DATA_BLOCK "DB_EmXcut_M203_SnapM201_HMI"
{ DB_Accessible_From_OPC_UA := 'FALSE' ;
 DB_Accessible_From_Webserver := 'FALSE' ;
 S7_Optimized_Access := 'FALSE' }
VERSION : 0.1
NON_RETAIN
   STRUCT
      tALM { ExternalWritable := 'False'} : Struct   // HMI Alarms
         tE { ExternalWritable := 'False'} : Struct   // Stopping faults
            xSpare_0 { ExternalWritable := 'False'} : Bool;
            xSpare_1 { ExternalWritable := 'False'} : Bool;
            xSpare_2 { ExternalWritable := 'False'} : Bool;
            xSpare_3 { ExternalWritable := 'False'} : Bool;
            xSpare_4 { ExternalWritable := 'False'} : Bool;
            xSpare_5 { ExternalWritable := 'False'} : Bool;
            xSpare_6 { ExternalWritable := 'False'} : Bool;
            xSpare_7 { ExternalWritable := 'False'} : Bool;
            xSpare_8 { ExternalWritable := 'False'} : Bool;
            xSpare_9 { ExternalWritable := 'False'} : Bool;
            xSpare_10 { ExternalWritable := 'False'} : Bool;
            xSpare_11 { ExternalWritable := 'False'} : Bool;
            xSpare_12 { ExternalWritable := 'False'} : Bool;
            xSpare_13 { ExternalWritable := 'False'} : Bool;
            xSpare_14 { ExternalWritable := 'False'} : Bool;
            xSpare_15 { ExternalWritable := 'False'} : Bool;
            xSpare_16 { ExternalWritable := 'False'} : Bool;
            xSpare_17 { ExternalWritable := 'False'} : Bool;
            xSpare_18 { ExternalWritable := 'False'} : Bool;
            xSpare_19 { ExternalWritable := 'False'} : Bool;
            xSpare_20 { ExternalWritable := 'False'} : Bool;
            xSpare_21 { ExternalWritable := 'False'} : Bool;
            xSpare_22 { ExternalWritable := 'False'} : Bool;
            xSpare_23 { ExternalWritable := 'False'} : Bool;
            xSpare_24 { ExternalWritable := 'False'} : Bool;
            xSpare_25 { ExternalWritable := 'False'} : Bool;
            xSpare_26 { ExternalWritable := 'False'} : Bool;
            xSpare_27 { ExternalWritable := 'False'} : Bool;
            xSpare_28 { ExternalWritable := 'False'} : Bool;
            xSpare_29 { ExternalWritable := 'False'} : Bool;
            xSpare_30 { ExternalWritable := 'False'} : Bool;
            xSpare_31 { ExternalWritable := 'False'} : Bool;
         END_STRUCT;
         tS { ExternalWritable := 'False'} : Struct   // Stopping faults
            xMachineNotReady { ExternalWritable := 'False'} : Bool;   // Machine not ready
            xQMProtection { ExternalWritable := 'False'} : Bool;   // A172QM1.Protection
            xSpare_2 { ExternalAccessible := 'False'; ExternalVisible := 'False'; ExternalWritable := 'False'} : Bool;
            xSpare_3 { ExternalAccessible := 'False'; ExternalVisible := 'False'; ExternalWritable := 'False'} : Bool;
            xSpare_4 { ExternalAccessible := 'False'; ExternalVisible := 'False'; ExternalWritable := 'False'} : Bool;
            xSpare_5 { ExternalAccessible := 'False'; ExternalVisible := 'False'; ExternalWritable := 'False'} : Bool;
            xSpare_6 { ExternalAccessible := 'False'; ExternalVisible := 'False'; ExternalWritable := 'False'} : Bool;
            xSpare_7 { ExternalAccessible := 'False'; ExternalVisible := 'False'; ExternalWritable := 'False'} : Bool;
            xSpare_8 { ExternalAccessible := 'False'; ExternalVisible := 'False'; ExternalWritable := 'False'} : Bool;
            xSpare_9 { ExternalAccessible := 'False'; ExternalVisible := 'False'; ExternalWritable := 'False'} : Bool;
            xSpare_10 { ExternalAccessible := 'False'; ExternalVisible := 'False'; ExternalWritable := 'False'} : Bool;
            xSpare_11 { ExternalAccessible := 'False'; ExternalVisible := 'False'; ExternalWritable := 'False'} : Bool;
            xSpare_12 { ExternalAccessible := 'False'; ExternalVisible := 'False'; ExternalWritable := 'False'} : Bool;
            xSpare_13 { ExternalAccessible := 'False'; ExternalVisible := 'False'; ExternalWritable := 'False'} : Bool;
            xSpare_14 { ExternalAccessible := 'False'; ExternalVisible := 'False'; ExternalWritable := 'False'} : Bool;
            xSpare_15 { ExternalAccessible := 'False'; ExternalVisible := 'False'; ExternalWritable := 'False'} : Bool;
            xSpare_16 { ExternalAccessible := 'False'; ExternalVisible := 'False'; ExternalWritable := 'False'} : Bool;
            xSpare_17 { ExternalAccessible := 'False'; ExternalVisible := 'False'; ExternalWritable := 'False'} : Bool;
            xSpare_18 { ExternalAccessible := 'False'; ExternalVisible := 'False'; ExternalWritable := 'False'} : Bool;
            xSpare_19 { ExternalAccessible := 'False'; ExternalVisible := 'False'; ExternalWritable := 'False'} : Bool;
            xSpare_20 { ExternalAccessible := 'False'; ExternalVisible := 'False'; ExternalWritable := 'False'} : Bool;
            xSpare_21 { ExternalAccessible := 'False'; ExternalVisible := 'False'; ExternalWritable := 'False'} : Bool;
            xSpare_22 { ExternalAccessible := 'False'; ExternalVisible := 'False'; ExternalWritable := 'False'} : Bool;
            xSpare_23 { ExternalAccessible := 'False'; ExternalVisible := 'False'; ExternalWritable := 'False'} : Bool;
            xSpare_24 { ExternalAccessible := 'False'; ExternalVisible := 'False'; ExternalWritable := 'False'} : Bool;
            xSpare_25 { ExternalAccessible := 'False'; ExternalVisible := 'False'; ExternalWritable := 'False'} : Bool;
            xSpare_26 { ExternalAccessible := 'False'; ExternalVisible := 'False'; ExternalWritable := 'False'} : Bool;
            xSpare_27 { ExternalAccessible := 'False'; ExternalVisible := 'False'; ExternalWritable := 'False'} : Bool;
            xSpare_28 { ExternalAccessible := 'False'; ExternalVisible := 'False'; ExternalWritable := 'False'} : Bool;
            xSpare_29 { ExternalAccessible := 'False'; ExternalVisible := 'False'; ExternalWritable := 'False'} : Bool;
            xSpare_30 { ExternalAccessible := 'False'; ExternalVisible := 'False'; ExternalWritable := 'False'} : Bool;
            xSpare_31 { ExternalAccessible := 'False'; ExternalVisible := 'False'; ExternalWritable := 'False'} : Bool;
         END_STRUCT;
         tF { ExternalAccessible := 'False'; ExternalVisible := 'False'; ExternalWritable := 'False'} : Struct   // Faults
            xSpare_0 { ExternalAccessible := 'False'; ExternalVisible := 'False'; ExternalWritable := 'False'} : Bool;
            xSpare_1 { ExternalAccessible := 'False'; ExternalVisible := 'False'; ExternalWritable := 'False'} : Bool;
            xSpare_2 { ExternalAccessible := 'False'; ExternalVisible := 'False'; ExternalWritable := 'False'} : Bool;
            xSpare_3 { ExternalAccessible := 'False'; ExternalVisible := 'False'; ExternalWritable := 'False'} : Bool;
            xSpare_4 { ExternalAccessible := 'False'; ExternalVisible := 'False'; ExternalWritable := 'False'} : Bool;
            xSpare_5 { ExternalAccessible := 'False'; ExternalVisible := 'False'; ExternalWritable := 'False'} : Bool;
            xSpare_6 { ExternalAccessible := 'False'; ExternalVisible := 'False'; ExternalWritable := 'False'} : Bool;
            xSpare_7 { ExternalAccessible := 'False'; ExternalVisible := 'False'; ExternalWritable := 'False'} : Bool;
            xSpare_8 { ExternalAccessible := 'False'; ExternalVisible := 'False'; ExternalWritable := 'False'} : Bool;
            xSpare_9 { ExternalAccessible := 'False'; ExternalVisible := 'False'; ExternalWritable := 'False'} : Bool;
            xSpare_10 { ExternalAccessible := 'False'; ExternalVisible := 'False'; ExternalWritable := 'False'} : Bool;
            xSpare_11 { ExternalAccessible := 'False'; ExternalVisible := 'False'; ExternalWritable := 'False'} : Bool;
            xSpare_12 { ExternalAccessible := 'False'; ExternalVisible := 'False'; ExternalWritable := 'False'} : Bool;
            xSpare_13 { ExternalAccessible := 'False'; ExternalVisible := 'False'; ExternalWritable := 'False'} : Bool;
            xSpare_14 { ExternalAccessible := 'False'; ExternalVisible := 'False'; ExternalWritable := 'False'} : Bool;
            xSpare_15 { ExternalAccessible := 'False'; ExternalVisible := 'False'; ExternalWritable := 'False'} : Bool;
            xSpare_16 { ExternalAccessible := 'False'; ExternalVisible := 'False'; ExternalWritable := 'False'} : Bool;
            xSpare_17 { ExternalAccessible := 'False'; ExternalVisible := 'False'; ExternalWritable := 'False'} : Bool;
            xSpare_18 { ExternalAccessible := 'False'; ExternalVisible := 'False'; ExternalWritable := 'False'} : Bool;
            xSpare_19 { ExternalAccessible := 'False'; ExternalVisible := 'False'; ExternalWritable := 'False'} : Bool;
            xSpare_20 { ExternalAccessible := 'False'; ExternalVisible := 'False'; ExternalWritable := 'False'} : Bool;
            xSpare_21 { ExternalAccessible := 'False'; ExternalVisible := 'False'; ExternalWritable := 'False'} : Bool;
            xSpare_22 { ExternalAccessible := 'False'; ExternalVisible := 'False'; ExternalWritable := 'False'} : Bool;
            xSpare_23 { ExternalAccessible := 'False'; ExternalVisible := 'False'; ExternalWritable := 'False'} : Bool;
            xSpare_24 { ExternalAccessible := 'False'; ExternalVisible := 'False'; ExternalWritable := 'False'} : Bool;
            xSpare_25 { ExternalAccessible := 'False'; ExternalVisible := 'False'; ExternalWritable := 'False'} : Bool;
            xSpare_26 { ExternalAccessible := 'False'; ExternalVisible := 'False'; ExternalWritable := 'False'} : Bool;
            xSpare_27 { ExternalAccessible := 'False'; ExternalVisible := 'False'; ExternalWritable := 'False'} : Bool;
            xSpare_28 { ExternalAccessible := 'False'; ExternalVisible := 'False'; ExternalWritable := 'False'} : Bool;
            xSpare_29 { ExternalAccessible := 'False'; ExternalVisible := 'False'; ExternalWritable := 'False'} : Bool;
            xSpare_30 { ExternalAccessible := 'False'; ExternalVisible := 'False'; ExternalWritable := 'False'} : Bool;
            xSpare_31 { ExternalAccessible := 'False'; ExternalVisible := 'False'; ExternalWritable := 'False'} : Bool;
         END_STRUCT;
         tW { ExternalAccessible := 'False'; ExternalVisible := 'False'; ExternalWritable := 'False'} : Struct   // Warnings
            xSpare_0 { ExternalAccessible := 'False'; ExternalVisible := 'False'; ExternalWritable := 'False'} : Bool;
            xSpare_1 { ExternalAccessible := 'False'; ExternalVisible := 'False'; ExternalWritable := 'False'} : Bool;
            xSpare_2 { ExternalAccessible := 'False'; ExternalVisible := 'False'; ExternalWritable := 'False'} : Bool;
            xSpare_3 { ExternalAccessible := 'False'; ExternalVisible := 'False'; ExternalWritable := 'False'} : Bool;
            xSpare_4 { ExternalAccessible := 'False'; ExternalVisible := 'False'; ExternalWritable := 'False'} : Bool;
            xSpare_5 { ExternalAccessible := 'False'; ExternalVisible := 'False'; ExternalWritable := 'False'} : Bool;
            xSpare_6 { ExternalAccessible := 'False'; ExternalVisible := 'False'; ExternalWritable := 'False'} : Bool;
            xSpare_7 { ExternalAccessible := 'False'; ExternalVisible := 'False'; ExternalWritable := 'False'} : Bool;
            xSpare_8 { ExternalAccessible := 'False'; ExternalVisible := 'False'; ExternalWritable := 'False'} : Bool;
            xSpare_9 { ExternalAccessible := 'False'; ExternalVisible := 'False'; ExternalWritable := 'False'} : Bool;
            xSpare_10 { ExternalAccessible := 'False'; ExternalVisible := 'False'; ExternalWritable := 'False'} : Bool;
            xSpare_11 { ExternalAccessible := 'False'; ExternalVisible := 'False'; ExternalWritable := 'False'} : Bool;
            xSpare_12 { ExternalAccessible := 'False'; ExternalVisible := 'False'; ExternalWritable := 'False'} : Bool;
            xSpare_13 { ExternalAccessible := 'False'; ExternalVisible := 'False'; ExternalWritable := 'False'} : Bool;
            xSpare_14 { ExternalAccessible := 'False'; ExternalVisible := 'False'; ExternalWritable := 'False'} : Bool;
            xSpare_15 { ExternalAccessible := 'False'; ExternalVisible := 'False'; ExternalWritable := 'False'} : Bool;
            xSpare_16 { ExternalAccessible := 'False'; ExternalVisible := 'False'; ExternalWritable := 'False'} : Bool;
            xSpare_17 { ExternalAccessible := 'False'; ExternalVisible := 'False'; ExternalWritable := 'False'} : Bool;
            xSpare_18 { ExternalAccessible := 'False'; ExternalVisible := 'False'; ExternalWritable := 'False'} : Bool;
            xSpare_19 { ExternalAccessible := 'False'; ExternalVisible := 'False'; ExternalWritable := 'False'} : Bool;
            xSpare_20 { ExternalAccessible := 'False'; ExternalVisible := 'False'; ExternalWritable := 'False'} : Bool;
            xSpare_21 { ExternalAccessible := 'False'; ExternalVisible := 'False'; ExternalWritable := 'False'} : Bool;
            xSpare_22 { ExternalAccessible := 'False'; ExternalVisible := 'False'; ExternalWritable := 'False'} : Bool;
            xSpare_23 { ExternalAccessible := 'False'; ExternalVisible := 'False'; ExternalWritable := 'False'} : Bool;
            xSpare_24 { ExternalAccessible := 'False'; ExternalVisible := 'False'; ExternalWritable := 'False'} : Bool;
            xSpare_25 { ExternalAccessible := 'False'; ExternalVisible := 'False'; ExternalWritable := 'False'} : Bool;
            xSpare_26 { ExternalAccessible := 'False'; ExternalVisible := 'False'; ExternalWritable := 'False'} : Bool;
            xSpare_27 { ExternalAccessible := 'False'; ExternalVisible := 'False'; ExternalWritable := 'False'} : Bool;
            xSpare_28 { ExternalAccessible := 'False'; ExternalVisible := 'False'; ExternalWritable := 'False'} : Bool;
            xSpare_29 { ExternalAccessible := 'False'; ExternalVisible := 'False'; ExternalWritable := 'False'} : Bool;
            xSpare_30 { ExternalAccessible := 'False'; ExternalVisible := 'False'; ExternalWritable := 'False'} : Bool;
            xSpare_31 { ExternalAccessible := 'False'; ExternalVisible := 'False'; ExternalWritable := 'False'} : Bool;
         END_STRUCT;
      END_STRUCT;
      tHMR { ExternalWritable := 'False'} : Struct   // HMI Read
         xSpare0 { ExternalWritable := 'False'} : Bool;   //
         xSpare1 { ExternalWritable := 'False'} : Bool;   //
         xSpare2 { ExternalWritable := 'False'} : Bool;
         xSpare3 { ExternalWritable := 'False'} : Bool;
         xSpare4 { ExternalWritable := 'False'} : Bool;
         xSpare5 { ExternalWritable := 'False'} : Bool;
         xSpare6 { ExternalWritable := 'False'} : Bool;
         xSpare7 { ExternalWritable := 'False'} : Bool;
         xSpare8 { ExternalWritable := 'False'} : Bool;
         xSpare9 { ExternalWritable := 'False'} : Bool;
         xSpare10 { ExternalWritable := 'False'} : Bool;
         xSpare11 { ExternalWritable := 'False'} : Bool;
         xSpare12 { ExternalWritable := 'False'} : Bool;
         xSpare13 { ExternalWritable := 'False'} : Bool;
         xSpare14 { ExternalWritable := 'False'} : Bool;
         xSpare15 { ExternalWritable := 'False'} : Bool;
         xSpare16 { ExternalWritable := 'False'} : Bool;
         xSpare17 { ExternalWritable := 'False'} : Bool;
         xSpare18 { ExternalWritable := 'False'} : Bool;
         xSpare19 { ExternalWritable := 'False'} : Bool;
         xSpare20 { ExternalWritable := 'False'} : Bool;
         xSpare21 { ExternalWritable := 'False'} : Bool;
         xSpare22 { ExternalWritable := 'False'} : Bool;
         xSpare23 { ExternalWritable := 'False'} : Bool;
         xSpare24 { ExternalWritable := 'False'} : Bool;
         xSpare25 { ExternalWritable := 'False'} : Bool;
         xSpare26 { ExternalWritable := 'False'} : Bool;
         xSpare27 { ExternalWritable := 'False'} : Bool;
         xSpare28 { ExternalWritable := 'False'} : Bool;
         xSpare29 { ExternalWritable := 'False'} : Bool;
         xSpare30 { ExternalWritable := 'False'} : Bool;
         xSpare31 { ExternalWritable := 'False'} : Bool;
         xSpare { ExternalWritable := 'False'} : Array[0..15] of Bool;
         iSpare0 { ExternalWritable := 'False'} : Int;
         iSpare1 { ExternalWritable := 'False'} : Int;
         iSpare2 { ExternalWritable := 'False'} : Int;
         iSpare3 { ExternalWritable := 'False'} : Int;
         iSpare4 { ExternalWritable := 'False'} : Int;
         iSpare5 { ExternalWritable := 'False'} : Int;
         iSpare6 { ExternalWritable := 'False'} : Int;
         iSpare7 { ExternalWritable := 'False'} : Int;
         iSpare8 { ExternalWritable := 'False'} : Int;
         iSpare9 { ExternalWritable := 'False'} : Int;
         iSpare10 { ExternalWritable := 'False'} : Int;
         iSpare11 { ExternalWritable := 'False'} : Int;
         iSpare12 { ExternalWritable := 'False'} : Int;
         iSpare13 { ExternalWritable := 'False'} : Int;
         iSpare14 { ExternalWritable := 'False'} : Int;
         iSpare15 { ExternalWritable := 'False'} : Int;
         iSpare16 { ExternalWritable := 'False'} : Int;
         dDistanceSnaproll_cmm { ExternalWritable := 'False'} : DInt;   // Distance from snaproll [mm/100] {mm/100|mm|x|x|M}
         dState { ExternalWritable := 'False'} : DInt;   // State  (1=No anomaly, 3=Run, 7=Anomaly) {x|x|x|x|O}
         dSpare2 { ExternalWritable := 'False'} : DInt;   //
         dSpare3 { ExternalWritable := 'False'} : DInt;
         dSpare4 { ExternalWritable := 'False'} : DInt;
         dSpare5 { ExternalWritable := 'False'} : DInt;
         dSpare6 { ExternalWritable := 'False'} : DInt;
         dSpare7 { ExternalWritable := 'False'} : DInt;
         dSpare8 { ExternalWritable := 'False'} : DInt;
         dSpare9 { ExternalWritable := 'False'} : DInt;
         dSpare10 { ExternalWritable := 'False'} : DInt;
         dSpare11 { ExternalWritable := 'False'} : DInt;
         dSpare12 { ExternalWritable := 'False'} : DInt;
         dSpare13 { ExternalWritable := 'False'} : DInt;
         dSpare14 { ExternalWritable := 'False'} : DInt;
         dSpare15 { ExternalWritable := 'False'} : DInt;
         rSpare0 { ExternalWritable := 'False'} : Real;
         rSpare1 { ExternalWritable := 'False'} : Real;
         rSpare2 { ExternalWritable := 'False'} : Real;
         rSpare3 { ExternalWritable := 'False'} : Real;
         rSpare4 { ExternalWritable := 'False'} : Real;
         rSpare5 { ExternalWritable := 'False'} : Real;
         rSpare6 { ExternalWritable := 'False'} : Real;
         rSpare7 { ExternalWritable := 'False'} : Real;
         rSpare8 { ExternalWritable := 'False'} : Real;
         tManCmd { ExternalWritable := 'False'} : Struct
            xSpare0 { ExternalWritable := 'False'} : Bool;   //
            xSpare1 { ExternalWritable := 'False'} : Bool;   //
            xSpare2 { ExternalWritable := 'False'} : Bool;
            xSpare3 { ExternalWritable := 'False'} : Bool;
            xSpare4 { ExternalWritable := 'False'} : Bool;
            xSpare5 { ExternalWritable := 'False'} : Bool;
            xSpare6 { ExternalWritable := 'False'} : Bool;
            xSpare7 { ExternalWritable := 'False'} : Bool;
            xSpare8 { ExternalWritable := 'False'} : Bool;
            xSpare9 { ExternalWritable := 'False'} : Bool;
            xSpare10 { ExternalWritable := 'False'} : Bool;
            xSpare11 { ExternalWritable := 'False'} : Bool;
            xSpare12 { ExternalWritable := 'False'} : Bool;
            xSpare13 { ExternalWritable := 'False'} : Bool;
            xSpare14 { ExternalWritable := 'False'} : Bool;
            xSpare15 { ExternalWritable := 'False'} : Bool;
            xSpare { ExternalWritable := 'False'} : Array[0..15] of Bool;
         END_STRUCT;
      END_STRUCT;
      tHMW : Struct   // HMI Write
         xSpare0 : Bool;   //
         xSpare1 : Bool;   //
         xSpare2 : Bool;   //
         xSpare3 : Bool;   //
         xSpare4 : Bool;   //
         xSpare5 : Bool;
         xSpare6 : Bool;
         xSpare7 : Bool;
         xSpare8 : Bool;   //
         xSpare9 : Bool;
         xSpare10 : Bool;
         xSpare11 : Bool;
         xSpare12 : Bool;
         xSpare13 : Bool;
         xSpare14 : Bool;   //
         xUpdateDistanceSnaproll : Bool;   // Update distance from snaproll {x|x|x|x|M}
         xSpare16 : Bool;   //
         xSpare17 : Bool;
         xSpare18 : Bool;
         xSpare19 : Bool;
         xSpare20 : Bool;
         xSpare21 : Bool;
         xSpare22 : Bool;
         xSpare23 : Bool;
         xSpare24 : Bool;
         xSpare25 : Bool;
         xSpare26 : Bool;
         xSpare27 : Bool;
         xSpare28 : Bool;
         xSpare29 : Bool;
         xSpare30 : Bool;
         xSpare31 : Bool;
         xSpare : Array[0..15] of Bool;
         iSpare0 : Int;
         iSpare1 : Int;
         iSpare2 : Int;
         iSpare3 : Int;
         iSpare4 : Int;
         iSpare5 : Int;
         iSpare6 : Int;
         iSpare7 : Int;
         iSpare8 : Int;
         iSpare9 : Int;
         iSpare10 : Int;
         iSpare11 : Int;
         iSpare12 : Int;
         iSpare13 : Int;
         iSpare14 : Int;
         iSpare15 : Int;
         iSpare16 : Int;
         dDistanceSnaproll_cmm : DInt;   // Distance from snaproll [mm/100] {mm/100|mm|1|70000|M}
         dSnapDuration_ms : DInt;   // Time snap in up position [ms] {ms|s|0|1|O}
         AccelerationDelay_ms : DInt;   // Acceleration delay [ms] {ms|s|0|1|O}
         dSpare3 : DInt;
         dSpare4 : DInt;
         dSpare5 : DInt;
         dSpare6 : DInt;
         dSpare7 : DInt;
         dSpare8 : DInt;
         dSpare9 : DInt;
         dSpare10 : DInt;
         dSpare11 : DInt;
         dSpare12 : DInt;
         dSpare13 : DInt;
         dSpare14 : DInt;
         dSpare15 : DInt;
         dSpare16 : DInt;
         rPlateLenght_mm : Real;   // Maximum plate lenght for contrast enabling [mm] {mm|mm|1|7000|O}
         rBreakPosOffset_mm : Real;   // BreakOffset [mm] {mm|mm|1|1000|O}
         rSpare2 : Real;
         rSpare3 : Real;
         rSpare4 : Real;
         rSpare5 : Real;
         rSpare6 : Real;
         rSpare7 : Real;
         rSpare8 : Real;
         tManCmd : Struct
            xSpare0 : Bool;
            xSpare1 : Bool;   //
            xSpare2 { ExternalWritable := 'False'} : Bool;
            xSpare3 { ExternalWritable := 'False'} : Bool;
            xSpare4 { ExternalWritable := 'False'} : Bool;
            xSpare5 { ExternalWritable := 'False'} : Bool;
            xSpare6 { ExternalWritable := 'False'} : Bool;
            xSpare7 { ExternalWritable := 'False'} : Bool;
            xSpare8 { ExternalWritable := 'False'} : Bool;
            xSpare9 { ExternalWritable := 'False'} : Bool;
            xSpare10 { ExternalWritable := 'False'} : Bool;
            xSpare11 { ExternalWritable := 'False'} : Bool;
            xSpare12 { ExternalWritable := 'False'} : Bool;
            xSpare13 { ExternalWritable := 'False'} : Bool;
            xSpare14 { ExternalWritable := 'False'} : Bool;
            xSpare15 { ExternalWritable := 'False'} : Bool;
            xSpare16 : Bool;
            xSpare17 : Bool;
            xSpare18 : Bool;
            xSpare19 : Bool;
            xSpare20 : Bool;
            xSpare21 : Bool;
            xSpare22 : Bool;
            xSpare23 : Bool;
            xSpare24 : Bool;
            xSpare25 : Bool;
            xSpare26 : Bool;
            xSpare27 : Bool;
            xSpare28 : Bool;
            xSpare29 : Bool;
            xSpare30 : Bool;
            xSpare31 : Bool;
         END_STRUCT;
      END_STRUCT;
   END_STRUCT;


BEGIN
   tHMW.tManCmd.xSpare0 := false;
   tHMW.tManCmd.xSpare1 := false;

END_DATA_BLOCK

DATA_BLOCK "DB_Oil_Manager_HMI"
{ DB_Accessible_From_OPC_UA := 'FALSE' ;
 DB_Accessible_From_Webserver := 'FALSE' ;
 S7_Optimized_Access := 'FALSE' }
VERSION : 0.1
   STRUCT
      tALM { ExternalWritable := 'False'} : Struct   // HMI Alarms
         tE { ExternalWritable := 'False'} : Struct   // Stopping faults
            xSpare_0 { ExternalWritable := 'False'} : Bool;
            xSpare_1 { ExternalWritable := 'False'} : Bool;
            xSpare_2 { ExternalWritable := 'False'} : Bool;
            xSpare_3 { ExternalWritable := 'False'} : Bool;
            xSpare_4 { ExternalWritable := 'False'} : Bool;
            xSpare_5 { ExternalWritable := 'False'} : Bool;
            xSpare_6 { ExternalWritable := 'False'} : Bool;
            xSpare_7 { ExternalWritable := 'False'} : Bool;
            xSpare_8 { ExternalWritable := 'False'} : Bool;
            xSpare_9 { ExternalWritable := 'False'} : Bool;
            xSpare_10 { ExternalWritable := 'False'} : Bool;
            xSpare_11 { ExternalWritable := 'False'} : Bool;
            xSpare_12 { ExternalWritable := 'False'} : Bool;
            xSpare_13 { ExternalWritable := 'False'} : Bool;
            xSpare_14 { ExternalWritable := 'False'} : Bool;
            xSpare_15 { ExternalWritable := 'False'} : Bool;
            xSpare_16 { ExternalWritable := 'False'} : Bool;
            xSpare_17 { ExternalWritable := 'False'} : Bool;
            xSpare_18 { ExternalWritable := 'False'} : Bool;
            xSpare_19 { ExternalWritable := 'False'} : Bool;
            xSpare_20 { ExternalWritable := 'False'} : Bool;
            xSpare_21 { ExternalWritable := 'False'} : Bool;
            xSpare_22 { ExternalWritable := 'False'} : Bool;
            xSpare_23 { ExternalWritable := 'False'} : Bool;
            xSpare_24 { ExternalWritable := 'False'} : Bool;
            xSpare_25 { ExternalWritable := 'False'} : Bool;
            xSpare_26 { ExternalWritable := 'False'} : Bool;
            xSpare_27 { ExternalWritable := 'False'} : Bool;
            xSpare_28 { ExternalWritable := 'False'} : Bool;
            xSpare_29 { ExternalWritable := 'False'} : Bool;
            xSpare_30 { ExternalWritable := 'False'} : Bool;
            xSpare_31 { ExternalWritable := 'False'} : Bool;
         END_STRUCT;
         tS { ExternalWritable := 'False'} : Struct   // Stopping faults machine
            xPowerSupplyControl { ExternalWritable := 'False'} : Bool;   // L+.Power supply control {X|X|X|X|O}
            xOilMinimumLevel { ExternalWritable := 'False'} : Bool;   // SL1.Oil at minimum {X|X|X|X|O}
            xTimeoutRefillOil { ExternalWritable := 'False'} : Bool;   // SL2.Timeout refill oil {X|X|X|X|O}
            xSensorMismatch { ExternalWritable := 'False'} : Bool;   // SL1/2.Sensor mismatch {X|X|X|X|O}
            xSpare_4 { ExternalAccessible := 'False'; ExternalVisible := 'False'; ExternalWritable := 'False'} : Bool;
            xSpare_5 { ExternalAccessible := 'False'; ExternalVisible := 'False'; ExternalWritable := 'False'} : Bool;
            xSpare_6 { ExternalAccessible := 'False'; ExternalVisible := 'False'; ExternalWritable := 'False'} : Bool;
            xSpare_7 { ExternalAccessible := 'False'; ExternalVisible := 'False'; ExternalWritable := 'False'} : Bool;
            xSpare_8 { ExternalAccessible := 'False'; ExternalVisible := 'False'; ExternalWritable := 'False'} : Bool;
            xSpare_9 { ExternalAccessible := 'False'; ExternalVisible := 'False'; ExternalWritable := 'False'} : Bool;
            xSpare_10 { ExternalAccessible := 'False'; ExternalVisible := 'False'; ExternalWritable := 'False'} : Bool;
            xSpare_11 { ExternalAccessible := 'False'; ExternalVisible := 'False'; ExternalWritable := 'False'} : Bool;
            xSpare_12 { ExternalAccessible := 'False'; ExternalVisible := 'False'; ExternalWritable := 'False'} : Bool;
            xSpare_13 { ExternalAccessible := 'False'; ExternalVisible := 'False'; ExternalWritable := 'False'} : Bool;
            xSpare_14 { ExternalAccessible := 'False'; ExternalVisible := 'False'; ExternalWritable := 'False'} : Bool;
            xSpare_15 { ExternalAccessible := 'False'; ExternalVisible := 'False'; ExternalWritable := 'False'} : Bool;
            xSpare_16 { ExternalAccessible := 'False'; ExternalVisible := 'False'; ExternalWritable := 'False'} : Bool;
            xSpare_17 { ExternalAccessible := 'False'; ExternalVisible := 'False'; ExternalWritable := 'False'} : Bool;
            xSpare_18 { ExternalAccessible := 'False'; ExternalVisible := 'False'; ExternalWritable := 'False'} : Bool;
            xSpare_19 { ExternalAccessible := 'False'; ExternalVisible := 'False'; ExternalWritable := 'False'} : Bool;
            xSpare_20 { ExternalAccessible := 'False'; ExternalVisible := 'False'; ExternalWritable := 'False'} : Bool;
            xSpare_21 { ExternalAccessible := 'False'; ExternalVisible := 'False'; ExternalWritable := 'False'} : Bool;
            xSpare_22 { ExternalAccessible := 'False'; ExternalVisible := 'False'; ExternalWritable := 'False'} : Bool;
            xSpare_23 { ExternalAccessible := 'False'; ExternalVisible := 'False'; ExternalWritable := 'False'} : Bool;
            xSpare_24 { ExternalAccessible := 'False'; ExternalVisible := 'False'; ExternalWritable := 'False'} : Bool;
            xSpare_25 { ExternalAccessible := 'False'; ExternalVisible := 'False'; ExternalWritable := 'False'} : Bool;
            xSpare_26 { ExternalAccessible := 'False'; ExternalVisible := 'False'; ExternalWritable := 'False'} : Bool;
            xSpare_27 { ExternalAccessible := 'False'; ExternalVisible := 'False'; ExternalWritable := 'False'} : Bool;
            xSpare_28 { ExternalAccessible := 'False'; ExternalVisible := 'False'; ExternalWritable := 'False'} : Bool;
            xSpare_29 { ExternalAccessible := 'False'; ExternalVisible := 'False'; ExternalWritable := 'False'} : Bool;
            xSpare_30 { ExternalAccessible := 'False'; ExternalVisible := 'False'; ExternalWritable := 'False'} : Bool;
            xSpare_31 { ExternalAccessible := 'False'; ExternalVisible := 'False'; ExternalWritable := 'False'} : Bool;
         END_STRUCT;
         tF { ExternalAccessible := 'False'; ExternalVisible := 'False'; ExternalWritable := 'False'} : Struct   // Faults
            xSpare_0 { ExternalAccessible := 'False'; ExternalVisible := 'False'; ExternalWritable := 'False'} : Bool;
            xSpare_1 { ExternalAccessible := 'False'; ExternalVisible := 'False'; ExternalWritable := 'False'} : Bool;
            xSpare_2 { ExternalAccessible := 'False'; ExternalVisible := 'False'; ExternalWritable := 'False'} : Bool;
            xSpare_3 { ExternalAccessible := 'False'; ExternalVisible := 'False'; ExternalWritable := 'False'} : Bool;
            xSpare_4 { ExternalAccessible := 'False'; ExternalVisible := 'False'; ExternalWritable := 'False'} : Bool;
            xSpare_5 { ExternalAccessible := 'False'; ExternalVisible := 'False'; ExternalWritable := 'False'} : Bool;
            xSpare_6 { ExternalAccessible := 'False'; ExternalVisible := 'False'; ExternalWritable := 'False'} : Bool;
            xSpare_7 { ExternalAccessible := 'False'; ExternalVisible := 'False'; ExternalWritable := 'False'} : Bool;
            xSpare_8 { ExternalAccessible := 'False'; ExternalVisible := 'False'; ExternalWritable := 'False'} : Bool;
            xSpare_9 { ExternalAccessible := 'False'; ExternalVisible := 'False'; ExternalWritable := 'False'} : Bool;
            xSpare_10 { ExternalAccessible := 'False'; ExternalVisible := 'False'; ExternalWritable := 'False'} : Bool;
            xSpare_11 { ExternalAccessible := 'False'; ExternalVisible := 'False'; ExternalWritable := 'False'} : Bool;
            xSpare_12 { ExternalAccessible := 'False'; ExternalVisible := 'False'; ExternalWritable := 'False'} : Bool;
            xSpare_13 { ExternalAccessible := 'False'; ExternalVisible := 'False'; ExternalWritable := 'False'} : Bool;
            xSpare_14 { ExternalAccessible := 'False'; ExternalVisible := 'False'; ExternalWritable := 'False'} : Bool;
            xSpare_15 { ExternalAccessible := 'False'; ExternalVisible := 'False'; ExternalWritable := 'False'} : Bool;
            xSpare_16 { ExternalAccessible := 'False'; ExternalVisible := 'False'; ExternalWritable := 'False'} : Bool;
            xSpare_17 { ExternalAccessible := 'False'; ExternalVisible := 'False'; ExternalWritable := 'False'} : Bool;
            xSpare_18 { ExternalAccessible := 'False'; ExternalVisible := 'False'; ExternalWritable := 'False'} : Bool;
            xSpare_19 { ExternalAccessible := 'False'; ExternalVisible := 'False'; ExternalWritable := 'False'} : Bool;
            xSpare_20 { ExternalAccessible := 'False'; ExternalVisible := 'False'; ExternalWritable := 'False'} : Bool;
            xSpare_21 { ExternalAccessible := 'False'; ExternalVisible := 'False'; ExternalWritable := 'False'} : Bool;
            xSpare_22 { ExternalAccessible := 'False'; ExternalVisible := 'False'; ExternalWritable := 'False'} : Bool;
            xSpare_23 { ExternalAccessible := 'False'; ExternalVisible := 'False'; ExternalWritable := 'False'} : Bool;
            xSpare_24 { ExternalAccessible := 'False'; ExternalVisible := 'False'; ExternalWritable := 'False'} : Bool;
            xSpare_25 { ExternalAccessible := 'False'; ExternalVisible := 'False'; ExternalWritable := 'False'} : Bool;
            xSpare_26 { ExternalAccessible := 'False'; ExternalVisible := 'False'; ExternalWritable := 'False'} : Bool;
            xSpare_27 { ExternalAccessible := 'False'; ExternalVisible := 'False'; ExternalWritable := 'False'} : Bool;
            xSpare_28 { ExternalAccessible := 'False'; ExternalVisible := 'False'; ExternalWritable := 'False'} : Bool;
            xSpare_29 { ExternalAccessible := 'False'; ExternalVisible := 'False'; ExternalWritable := 'False'} : Bool;
            xSpare_30 { ExternalAccessible := 'False'; ExternalVisible := 'False'; ExternalWritable := 'False'} : Bool;
            xSpare_31 { ExternalAccessible := 'False'; ExternalVisible := 'False'; ExternalWritable := 'False'} : Bool;
         END_STRUCT;
         tW { ExternalAccessible := 'False'; ExternalVisible := 'False'; ExternalWritable := 'False'} : Struct   // Warnings
            xSpare_0 { ExternalAccessible := 'False'; ExternalVisible := 'False'; ExternalWritable := 'False'} : Bool;
            xSpare_1 { ExternalAccessible := 'False'; ExternalVisible := 'False'; ExternalWritable := 'False'} : Bool;
            xSpare_2 { ExternalAccessible := 'False'; ExternalVisible := 'False'; ExternalWritable := 'False'} : Bool;
            xSpare_3 { ExternalAccessible := 'False'; ExternalVisible := 'False'; ExternalWritable := 'False'} : Bool;
            xSpare_4 { ExternalAccessible := 'False'; ExternalVisible := 'False'; ExternalWritable := 'False'} : Bool;
            xSpare_5 { ExternalAccessible := 'False'; ExternalVisible := 'False'; ExternalWritable := 'False'} : Bool;
            xSpare_6 { ExternalAccessible := 'False'; ExternalVisible := 'False'; ExternalWritable := 'False'} : Bool;
            xSpare_7 { ExternalAccessible := 'False'; ExternalVisible := 'False'; ExternalWritable := 'False'} : Bool;
            xSpare_8 { ExternalAccessible := 'False'; ExternalVisible := 'False'; ExternalWritable := 'False'} : Bool;
            xSpare_9 { ExternalAccessible := 'False'; ExternalVisible := 'False'; ExternalWritable := 'False'} : Bool;
            xSpare_10 { ExternalAccessible := 'False'; ExternalVisible := 'False'; ExternalWritable := 'False'} : Bool;
            xSpare_11 { ExternalAccessible := 'False'; ExternalVisible := 'False'; ExternalWritable := 'False'} : Bool;
            xSpare_12 { ExternalAccessible := 'False'; ExternalVisible := 'False'; ExternalWritable := 'False'} : Bool;
            xSpare_13 { ExternalAccessible := 'False'; ExternalVisible := 'False'; ExternalWritable := 'False'} : Bool;
            xSpare_14 { ExternalAccessible := 'False'; ExternalVisible := 'False'; ExternalWritable := 'False'} : Bool;
            xSpare_15 { ExternalAccessible := 'False'; ExternalVisible := 'False'; ExternalWritable := 'False'} : Bool;
            xSpare_16 { ExternalAccessible := 'False'; ExternalVisible := 'False'; ExternalWritable := 'False'} : Bool;
            xSpare_17 { ExternalAccessible := 'False'; ExternalVisible := 'False'; ExternalWritable := 'False'} : Bool;
            xSpare_18 { ExternalAccessible := 'False'; ExternalVisible := 'False'; ExternalWritable := 'False'} : Bool;
            xSpare_19 { ExternalAccessible := 'False'; ExternalVisible := 'False'; ExternalWritable := 'False'} : Bool;
            xSpare_20 { ExternalAccessible := 'False'; ExternalVisible := 'False'; ExternalWritable := 'False'} : Bool;
            xSpare_21 { ExternalAccessible := 'False'; ExternalVisible := 'False'; ExternalWritable := 'False'} : Bool;
            xSpare_22 { ExternalAccessible := 'False'; ExternalVisible := 'False'; ExternalWritable := 'False'} : Bool;
            xSpare_23 { ExternalAccessible := 'False'; ExternalVisible := 'False'; ExternalWritable := 'False'} : Bool;
            xSpare_24 { ExternalAccessible := 'False'; ExternalVisible := 'False'; ExternalWritable := 'False'} : Bool;
            xSpare_25 { ExternalAccessible := 'False'; ExternalVisible := 'False'; ExternalWritable := 'False'} : Bool;
            xSpare_26 { ExternalAccessible := 'False'; ExternalVisible := 'False'; ExternalWritable := 'False'} : Bool;
            xSpare_27 { ExternalAccessible := 'False'; ExternalVisible := 'False'; ExternalWritable := 'False'} : Bool;
            xSpare_28 { ExternalAccessible := 'False'; ExternalVisible := 'False'; ExternalWritable := 'False'} : Bool;
            xSpare_29 { ExternalAccessible := 'False'; ExternalVisible := 'False'; ExternalWritable := 'False'} : Bool;
            xSpare_30 { ExternalAccessible := 'False'; ExternalVisible := 'False'; ExternalWritable := 'False'} : Bool;
            xSpare_31 { ExternalAccessible := 'False'; ExternalVisible := 'False'; ExternalWritable := 'False'} : Bool;
         END_STRUCT;
      END_STRUCT;
      tHMR { ExternalWritable := 'False'} : Struct   // HMI Read
         xOilAtMin { ExternalWritable := 'False'} : Bool;   // Oil at minimum {X|X|X|X|O}
         xOilAtMax { ExternalWritable := 'False'} : Bool;   // Oil at maximum {X|X|X|X|O}
         xSpare2 { ExternalWritable := 'False'} : Bool;
         xSpare3 { ExternalWritable := 'False'} : Bool;
         xSpare4 { ExternalWritable := 'False'} : Bool;
         xSpare5 { ExternalWritable := 'False'} : Bool;
         xSpare6 { ExternalWritable := 'False'} : Bool;
         xSpare7 { ExternalWritable := 'False'} : Bool;
         xSpare8 { ExternalWritable := 'False'} : Bool;
         xSpare9 { ExternalWritable := 'False'} : Bool;
         xSpare10 { ExternalWritable := 'False'} : Bool;
         xSpare11 { ExternalWritable := 'False'} : Bool;
         xSpare12 { ExternalWritable := 'False'} : Bool;
         xSpare13 { ExternalWritable := 'False'} : Bool;
         xManualCommandEnabled { ExternalWritable := 'False'} : Bool;   // Manual Command enabled {x|x|x|x|O}
         xSpare15 { ExternalWritable := 'False'} : Bool;
         xSpare16 { ExternalWritable := 'False'} : Bool;
         xSpare17 { ExternalWritable := 'False'} : Bool;
         xSpare18 { ExternalWritable := 'False'} : Bool;
         xSpare19 { ExternalWritable := 'False'} : Bool;
         xSpare20 { ExternalWritable := 'False'} : Bool;
         xSpare21 { ExternalWritable := 'False'} : Bool;
         xSpare22 { ExternalWritable := 'False'} : Bool;
         xSpare23 { ExternalWritable := 'False'} : Bool;
         xSpare24 { ExternalWritable := 'False'} : Bool;
         xSpare25 { ExternalWritable := 'False'} : Bool;
         xSpare26 { ExternalWritable := 'False'} : Bool;
         xSpare27 { ExternalWritable := 'False'} : Bool;
         xSpare28 { ExternalWritable := 'False'} : Bool;
         xSpare29 { ExternalWritable := 'False'} : Bool;
         xSpare30 { ExternalWritable := 'False'} : Bool;
         xSpare31 { ExternalWritable := 'False'} : Bool;
         xSpare { ExternalWritable := 'False'} : Array[0..15] of Bool;
         iSpare0 { ExternalWritable := 'False'} : Int;
         iSpare1 { ExternalWritable := 'False'} : Int;
         iSpare2 { ExternalWritable := 'False'} : Int;
         iSpare3 { ExternalWritable := 'False'} : Int;
         iSpare4 { ExternalWritable := 'False'} : Int;
         iSpare5 { ExternalWritable := 'False'} : Int;
         iSpare6 { ExternalWritable := 'False'} : Int;
         iSpare7 { ExternalWritable := 'False'} : Int;
         iSpare8 { ExternalWritable := 'False'} : Int;
         iSpare9 { ExternalWritable := 'False'} : Int;
         iSpare10 { ExternalWritable := 'False'} : Int;
         iSpare11 { ExternalWritable := 'False'} : Int;
         iSpare12 { ExternalWritable := 'False'} : Int;
         iSpare13 { ExternalWritable := 'False'} : Int;
         iSpare14 { ExternalWritable := 'False'} : Int;
         iSpare15 { ExternalWritable := 'False'} : Int;
         iSpare16 { ExternalWritable := 'False'} : Int;
         dStatus { ExternalWritable := 'False'} : DInt;   // Status (1=Idle 3=Run 7=Anomaly) {X|X|X|X|O}
         dSpare1 { ExternalWritable := 'False'} : DInt;
         dSpare2 { ExternalWritable := 'False'} : DInt;
         dSpare3 { ExternalWritable := 'False'} : DInt;
         dSpare4 { ExternalWritable := 'False'} : DInt;
         dSpare5 { ExternalWritable := 'False'} : DInt;
         dSpare6 { ExternalWritable := 'False'} : DInt;
         dSpare7 { ExternalWritable := 'False'} : DInt;
         dSpare8 { ExternalWritable := 'False'} : DInt;
         dSpare9 { ExternalWritable := 'False'} : DInt;
         dSpare10 { ExternalWritable := 'False'} : DInt;
         dSpare11 { ExternalWritable := 'False'} : DInt;
         dSpare12 { ExternalWritable := 'False'} : DInt;
         dSpare13 { ExternalWritable := 'False'} : DInt;
         dSpare14 { ExternalWritable := 'False'} : DInt;
         dSpare15 { ExternalWritable := 'False'} : DInt;
         rSpare0 { ExternalWritable := 'False'} : Real;
         rSpare1 { ExternalWritable := 'False'} : Real;
         rSpare2 { ExternalWritable := 'False'} : Real;
         rSpare3 { ExternalWritable := 'False'} : Real;
         rSpare4 { ExternalWritable := 'False'} : Real;
         rSpare5 { ExternalWritable := 'False'} : Real;
         rSpare6 { ExternalWritable := 'False'} : Real;
         rSpare7 { ExternalWritable := 'False'} : Real;
         rSpare8 { ExternalWritable := 'False'} : Real;
         tManCmd { ExternalWritable := 'False'} : Struct
            xFillTank { ExternalWritable := 'False'} : Bool;   // Fill tank {x|x|x|x|O}
            xSpare1 { ExternalWritable := 'False'} : Bool;
            xSpare2 { ExternalWritable := 'False'} : Bool;
            xSpare3 { ExternalWritable := 'False'} : Bool;
            xSpare4 { ExternalWritable := 'False'} : Bool;
            xSpare5 { ExternalWritable := 'False'} : Bool;
            xSpare6 { ExternalWritable := 'False'} : Bool;
            xSpare7 { ExternalWritable := 'False'} : Bool;
            xSpare8 { ExternalWritable := 'False'} : Bool;
            xSpare9 { ExternalWritable := 'False'} : Bool;
            xSpare10 { ExternalWritable := 'False'} : Bool;
            xSpare11 { ExternalWritable := 'False'} : Bool;
            xSpare12 { ExternalWritable := 'False'} : Bool;
            xSpare13 { ExternalWritable := 'False'} : Bool;
            xSpare14 { ExternalWritable := 'False'} : Bool;
            xSpare15 { ExternalWritable := 'False'} : Bool;
            xSpare { ExternalWritable := 'False'} : Array[0..15] of Bool;
         END_STRUCT;
      END_STRUCT;
      tHMW : Struct   // HMI Write
         xSpare0 : Bool;   //
         xSpare1 : Bool;
         xSpare2 : Bool;
         xSpare3 : Bool;
         xSpare4 : Bool;
         xSpare5 : Bool;
         xSpare6 : Bool;
         xSpare7 : Bool;
         xSpare8 : Bool;
         xSpare9 : Bool;
         xSpare10 : Bool;   //
         xSpare11 : Bool;
         xSpare12 : Bool;
         xSpare13 : Bool;
         xEnableManualCommand : Bool;   // Enable Disable Manual command {x|x|x|x|O}
         xSpare15 : Bool;
         xSpare16 : Bool;
         xSpare17 : Bool;
         xSpare18 : Bool;
         xSpare19 : Bool;
         xSpare20 : Bool;
         xSpare21 : Bool;
         xSpare22 : Bool;
         xSpare23 : Bool;
         xSpare24 : Bool;
         xSpare25 : Bool;
         xSpare26 : Bool;
         xSpare27 : Bool;
         xSpare28 : Bool;
         xSpare29 : Bool;
         xSpare30 : Bool;
         xSpare31 : Bool;
         xSpare : Array[0..15] of Bool;
         iSpare0 : Int;
         iSpare1 : Int;
         iSpare2 : Int;
         iSpare3 : Int;
         iSpare4 : Int;
         iSpare5 : Int;
         iSpare6 : Int;
         iSpare7 : Int;
         iSpare8 : Int;
         iSpare9 : Int;
         iSpare10 : Int;
         iSpare11 : Int;
         iSpare12 : Int;
         iSpare13 : Int;
         iSpare14 : Int;
         iSpare15 : Int;
         iSpare16 : Int;
         dSpare0 : DInt;   //
         dSpare1 : DInt;
         dSpare2 : DInt;
         dSpare3 : DInt;
         dSpare4 : DInt;
         dSpare5 : DInt;
         dSpare6 : DInt;
         dSpare7 : DInt;
         dSpare8 : DInt;
         dSpare9 : DInt;
         dSpare10 : DInt;
         dSpare11 : DInt;
         dSpare12 : DInt;
         dSpare13 : DInt;
         dSpare14 : DInt;
         dSpare15 : DInt;
         dSpare16 : DInt;
         rSpare0 : Real;
         rSpare1 : Real;
         rSpare2 : Real;
         rSpare3 : Real;
         rSpare4 : Real;
         rSpare5 : Real;
         rSpare6 : Real;
         rSpare7 : Real;
         rSpare8 : Real;
         tManCmd : Struct
            xFillTank : Bool;   // Fill tank {x|x|x|x|O}
            xSpare1 : Bool;
            xSpare2 { ExternalWritable := 'False'} : Bool;
            xSpare3 { ExternalWritable := 'False'} : Bool;
            xSpare4 { ExternalWritable := 'False'} : Bool;
            xSpare5 { ExternalWritable := 'False'} : Bool;
            xSpare6 { ExternalWritable := 'False'} : Bool;
            xSpare7 { ExternalWritable := 'False'} : Bool;
            xSpare8 { ExternalWritable := 'False'} : Bool;
            xSpare9 { ExternalWritable := 'False'} : Bool;
            xSpare10 { ExternalWritable := 'False'} : Bool;
            xSpare11 { ExternalWritable := 'False'} : Bool;
            xSpare12 { ExternalWritable := 'False'} : Bool;
            xSpare13 { ExternalWritable := 'False'} : Bool;
            xSpare14 { ExternalWritable := 'False'} : Bool;
            xSpare15 { ExternalWritable := 'False'} : Bool;
            xSpare16 : Bool;
            xSpare17 : Bool;
            xSpare18 : Bool;
            xSpare19 : Bool;
            xSpare20 : Bool;
            xSpare21 : Bool;
            xSpare22 : Bool;
            xSpare23 : Bool;
            xSpare24 : Bool;
            xSpare25 : Bool;
            xSpare26 : Bool;
            xSpare27 : Bool;
            xSpare28 : Bool;
            xSpare29 : Bool;
            xSpare30 : Bool;
            xSpare31 : Bool;
         END_STRUCT;
      END_STRUCT;
   END_STRUCT;


BEGIN

END_DATA_BLOCK

DATA_BLOCK "DB_WANDER_HMI"
{ DB_Accessible_From_OPC_UA := 'FALSE' ;
 DB_Accessible_From_Webserver := 'FALSE' ;
 S7_Optimized_Access := 'FALSE' }
VERSION : 0.1
NON_RETAIN
   STRUCT
      tALM { ExternalWritable := 'False'} : Struct   // HMI Alarms
         tE { ExternalWritable := 'False'} : Struct   // Stopping faults
            xSpare_0 { ExternalWritable := 'False'} : Bool;
            xSpare_1 { ExternalWritable := 'False'} : Bool;
            xSpare_2 { ExternalWritable := 'False'} : Bool;
            xSpare_3 { ExternalWritable := 'False'} : Bool;
            xSpare_4 { ExternalWritable := 'False'} : Bool;
            xSpare_5 { ExternalWritable := 'False'} : Bool;
            xSpare_6 { ExternalWritable := 'False'} : Bool;
            xSpare_7 { ExternalWritable := 'False'} : Bool;
            xSpare_8 { ExternalWritable := 'False'} : Bool;
            xSpare_9 { ExternalWritable := 'False'} : Bool;
            xSpare_10 { ExternalWritable := 'False'} : Bool;
            xSpare_11 { ExternalWritable := 'False'} : Bool;
            xSpare_12 { ExternalWritable := 'False'} : Bool;
            xSpare_13 { ExternalWritable := 'False'} : Bool;
            xSpare_14 { ExternalWritable := 'False'} : Bool;
            xSpare_15 { ExternalWritable := 'False'} : Bool;
            xSpare_16 { ExternalWritable := 'False'} : Bool;
            xSpare_17 { ExternalWritable := 'False'} : Bool;
            xSpare_18 { ExternalWritable := 'False'} : Bool;
            xSpare_19 { ExternalWritable := 'False'} : Bool;
            xSpare_20 { ExternalWritable := 'False'} : Bool;
            xSpare_21 { ExternalWritable := 'False'} : Bool;
            xSpare_22 { ExternalWritable := 'False'} : Bool;
            xSpare_23 { ExternalWritable := 'False'} : Bool;
            xSpare_24 { ExternalWritable := 'False'} : Bool;
            xSpare_25 { ExternalWritable := 'False'} : Bool;
            xSpare_26 { ExternalWritable := 'False'} : Bool;
            xSpare_27 { ExternalWritable := 'False'} : Bool;
            xSpare_28 { ExternalWritable := 'False'} : Bool;
            xSpare_29 { ExternalWritable := 'False'} : Bool;
            xSpare_30 { ExternalWritable := 'False'} : Bool;
            xSpare_31 { ExternalWritable := 'False'} : Bool;
         END_STRUCT;
         tS { ExternalWritable := 'False'} : Struct   // Stopping faults
            xCameraNotConnected { ExternalWritable := 'False'} : Bool;   // Camera system not connected
            xSendError { ExternalWritable := 'False'} : Bool;   // Sending data error
            xSendTimeout { ExternalWritable := 'False'} : Bool;   // Sending data timeout
            xRecvTimeout { ExternalWritable := 'False'} : Bool;   // Receiving data timeout
            xWanderOutLimits { ExternalWritable := 'False'} : Bool;   // Wander outside limits
            xCameraInError { ExternalWritable := 'False'} : Bool;   // Camera system in error
            xSpare_6 { ExternalAccessible := 'False'; ExternalVisible := 'False'; ExternalWritable := 'False'} : Bool;
            xSpare_7 { ExternalAccessible := 'False'; ExternalVisible := 'False'; ExternalWritable := 'False'} : Bool;
            xSpare_8 { ExternalAccessible := 'False'; ExternalVisible := 'False'; ExternalWritable := 'False'} : Bool;
            xSpare_9 { ExternalAccessible := 'False'; ExternalVisible := 'False'; ExternalWritable := 'False'} : Bool;
            xSpare_10 { ExternalAccessible := 'False'; ExternalVisible := 'False'; ExternalWritable := 'False'} : Bool;
            xSpare_11 { ExternalAccessible := 'False'; ExternalVisible := 'False'; ExternalWritable := 'False'} : Bool;
            xSpare_12 { ExternalAccessible := 'False'; ExternalVisible := 'False'; ExternalWritable := 'False'} : Bool;
            xSpare_13 { ExternalAccessible := 'False'; ExternalVisible := 'False'; ExternalWritable := 'False'} : Bool;
            xSpare_14 { ExternalAccessible := 'False'; ExternalVisible := 'False'; ExternalWritable := 'False'} : Bool;
            xSpare_15 { ExternalAccessible := 'False'; ExternalVisible := 'False'; ExternalWritable := 'False'} : Bool;
            xSpare_16 { ExternalAccessible := 'False'; ExternalVisible := 'False'; ExternalWritable := 'False'} : Bool;
            xSpare_17 { ExternalAccessible := 'False'; ExternalVisible := 'False'; ExternalWritable := 'False'} : Bool;
            xSpare_18 { ExternalAccessible := 'False'; ExternalVisible := 'False'; ExternalWritable := 'False'} : Bool;
            xSpare_19 { ExternalAccessible := 'False'; ExternalVisible := 'False'; ExternalWritable := 'False'} : Bool;
            xSpare_20 { ExternalAccessible := 'False'; ExternalVisible := 'False'; ExternalWritable := 'False'} : Bool;
            xSpare_21 { ExternalAccessible := 'False'; ExternalVisible := 'False'; ExternalWritable := 'False'} : Bool;
            xSpare_22 { ExternalAccessible := 'False'; ExternalVisible := 'False'; ExternalWritable := 'False'} : Bool;
            xSpare_23 { ExternalAccessible := 'False'; ExternalVisible := 'False'; ExternalWritable := 'False'} : Bool;
            xSpare_24 { ExternalAccessible := 'False'; ExternalVisible := 'False'; ExternalWritable := 'False'} : Bool;
            xSpare_25 { ExternalAccessible := 'False'; ExternalVisible := 'False'; ExternalWritable := 'False'} : Bool;
            xSpare_26 { ExternalAccessible := 'False'; ExternalVisible := 'False'; ExternalWritable := 'False'} : Bool;
            xSpare_27 { ExternalAccessible := 'False'; ExternalVisible := 'False'; ExternalWritable := 'False'} : Bool;
            xSpare_28 { ExternalAccessible := 'False'; ExternalVisible := 'False'; ExternalWritable := 'False'} : Bool;
            xSpare_29 { ExternalAccessible := 'False'; ExternalVisible := 'False'; ExternalWritable := 'False'} : Bool;
            xSpare_30 { ExternalAccessible := 'False'; ExternalVisible := 'False'; ExternalWritable := 'False'} : Bool;
            xSpare_31 { ExternalAccessible := 'False'; ExternalVisible := 'False'; ExternalWritable := 'False'} : Bool;
         END_STRUCT;
         tF { ExternalWritable := 'False'} : Struct   // Faults
            xSpare_0 { ExternalAccessible := 'False'; ExternalVisible := 'False'; ExternalWritable := 'False'} : Bool;
            xSpare_1 { ExternalAccessible := 'False'; ExternalVisible := 'False'; ExternalWritable := 'False'} : Bool;
            xSpare_2 { ExternalAccessible := 'False'; ExternalVisible := 'False'; ExternalWritable := 'False'} : Bool;
            xSpare_3 { ExternalAccessible := 'False'; ExternalVisible := 'False'; ExternalWritable := 'False'} : Bool;
            xSpare_4 { ExternalAccessible := 'False'; ExternalVisible := 'False'; ExternalWritable := 'False'} : Bool;
            xSpare_5 { ExternalAccessible := 'False'; ExternalVisible := 'False'; ExternalWritable := 'False'} : Bool;
            xSpare_6 { ExternalAccessible := 'False'; ExternalVisible := 'False'; ExternalWritable := 'False'} : Bool;
            xSpare_7 { ExternalAccessible := 'False'; ExternalVisible := 'False'; ExternalWritable := 'False'} : Bool;
            xSpare_8 { ExternalAccessible := 'False'; ExternalVisible := 'False'; ExternalWritable := 'False'} : Bool;
            xSpare_9 { ExternalAccessible := 'False'; ExternalVisible := 'False'; ExternalWritable := 'False'} : Bool;
            xSpare_10 { ExternalAccessible := 'False'; ExternalVisible := 'False'; ExternalWritable := 'False'} : Bool;
            xSpare_11 { ExternalAccessible := 'False'; ExternalVisible := 'False'; ExternalWritable := 'False'} : Bool;
            xSpare_12 { ExternalAccessible := 'False'; ExternalVisible := 'False'; ExternalWritable := 'False'} : Bool;
            xSpare_13 { ExternalAccessible := 'False'; ExternalVisible := 'False'; ExternalWritable := 'False'} : Bool;
            xSpare_14 { ExternalAccessible := 'False'; ExternalVisible := 'False'; ExternalWritable := 'False'} : Bool;
            xSpare_15 { ExternalAccessible := 'False'; ExternalVisible := 'False'; ExternalWritable := 'False'} : Bool;
            xSpare_16 { ExternalAccessible := 'False'; ExternalVisible := 'False'; ExternalWritable := 'False'} : Bool;
            xSpare_17 { ExternalAccessible := 'False'; ExternalVisible := 'False'; ExternalWritable := 'False'} : Bool;
            xSpare_18 { ExternalAccessible := 'False'; ExternalVisible := 'False'; ExternalWritable := 'False'} : Bool;
            xSpare_19 { ExternalAccessible := 'False'; ExternalVisible := 'False'; ExternalWritable := 'False'} : Bool;
            xSpare_20 { ExternalAccessible := 'False'; ExternalVisible := 'False'; ExternalWritable := 'False'} : Bool;
            xSpare_21 { ExternalAccessible := 'False'; ExternalVisible := 'False'; ExternalWritable := 'False'} : Bool;
            xSpare_22 { ExternalAccessible := 'False'; ExternalVisible := 'False'; ExternalWritable := 'False'} : Bool;
            xSpare_23 { ExternalAccessible := 'False'; ExternalVisible := 'False'; ExternalWritable := 'False'} : Bool;
            xSpare_24 { ExternalAccessible := 'False'; ExternalVisible := 'False'; ExternalWritable := 'False'} : Bool;
            xSpare_25 { ExternalAccessible := 'False'; ExternalVisible := 'False'; ExternalWritable := 'False'} : Bool;
            xSpare_26 { ExternalAccessible := 'False'; ExternalVisible := 'False'; ExternalWritable := 'False'} : Bool;
            xSpare_27 { ExternalAccessible := 'False'; ExternalVisible := 'False'; ExternalWritable := 'False'} : Bool;
            xSpare_28 { ExternalAccessible := 'False'; ExternalVisible := 'False'; ExternalWritable := 'False'} : Bool;
            xSpare_29 { ExternalAccessible := 'False'; ExternalVisible := 'False'; ExternalWritable := 'False'} : Bool;
            xSpare_30 { ExternalAccessible := 'False'; ExternalVisible := 'False'; ExternalWritable := 'False'} : Bool;
            xSpare_31 { ExternalAccessible := 'False'; ExternalVisible := 'False'; ExternalWritable := 'False'} : Bool;
         END_STRUCT;
         tW { ExternalAccessible := 'False'; ExternalVisible := 'False'; ExternalWritable := 'False'} : Struct   // Warnings
            xSpare_0 { ExternalAccessible := 'False'; ExternalVisible := 'False'; ExternalWritable := 'False'} : Bool;
            xSpare_1 { ExternalAccessible := 'False'; ExternalVisible := 'False'; ExternalWritable := 'False'} : Bool;
            xSpare_2 { ExternalAccessible := 'False'; ExternalVisible := 'False'; ExternalWritable := 'False'} : Bool;
            xSpare_3 { ExternalAccessible := 'False'; ExternalVisible := 'False'; ExternalWritable := 'False'} : Bool;
            xSpare_4 { ExternalAccessible := 'False'; ExternalVisible := 'False'; ExternalWritable := 'False'} : Bool;
            xSpare_5 { ExternalAccessible := 'False'; ExternalVisible := 'False'; ExternalWritable := 'False'} : Bool;
            xSpare_6 { ExternalAccessible := 'False'; ExternalVisible := 'False'; ExternalWritable := 'False'} : Bool;
            xSpare_7 { ExternalAccessible := 'False'; ExternalVisible := 'False'; ExternalWritable := 'False'} : Bool;
            xSpare_8 { ExternalAccessible := 'False'; ExternalVisible := 'False'; ExternalWritable := 'False'} : Bool;
            xSpare_9 { ExternalAccessible := 'False'; ExternalVisible := 'False'; ExternalWritable := 'False'} : Bool;
            xSpare_10 { ExternalAccessible := 'False'; ExternalVisible := 'False'; ExternalWritable := 'False'} : Bool;
            xSpare_11 { ExternalAccessible := 'False'; ExternalVisible := 'False'; ExternalWritable := 'False'} : Bool;
            xSpare_12 { ExternalAccessible := 'False'; ExternalVisible := 'False'; ExternalWritable := 'False'} : Bool;
            xSpare_13 { ExternalAccessible := 'False'; ExternalVisible := 'False'; ExternalWritable := 'False'} : Bool;
            xSpare_14 { ExternalAccessible := 'False'; ExternalVisible := 'False'; ExternalWritable := 'False'} : Bool;
            xSpare_15 { ExternalAccessible := 'False'; ExternalVisible := 'False'; ExternalWritable := 'False'} : Bool;
            xSpare_16 { ExternalAccessible := 'False'; ExternalVisible := 'False'; ExternalWritable := 'False'} : Bool;
            xSpare_17 { ExternalAccessible := 'False'; ExternalVisible := 'False'; ExternalWritable := 'False'} : Bool;
            xSpare_18 { ExternalAccessible := 'False'; ExternalVisible := 'False'; ExternalWritable := 'False'} : Bool;
            xSpare_19 { ExternalAccessible := 'False'; ExternalVisible := 'False'; ExternalWritable := 'False'} : Bool;
            xSpare_20 { ExternalAccessible := 'False'; ExternalVisible := 'False'; ExternalWritable := 'False'} : Bool;
            xSpare_21 { ExternalAccessible := 'False'; ExternalVisible := 'False'; ExternalWritable := 'False'} : Bool;
            xSpare_22 { ExternalAccessible := 'False'; ExternalVisible := 'False'; ExternalWritable := 'False'} : Bool;
            xSpare_23 { ExternalAccessible := 'False'; ExternalVisible := 'False'; ExternalWritable := 'False'} : Bool;
            xSpare_24 { ExternalAccessible := 'False'; ExternalVisible := 'False'; ExternalWritable := 'False'} : Bool;
            xSpare_25 { ExternalAccessible := 'False'; ExternalVisible := 'False'; ExternalWritable := 'False'} : Bool;
            xSpare_26 { ExternalAccessible := 'False'; ExternalVisible := 'False'; ExternalWritable := 'False'} : Bool;
            xSpare_27 { ExternalAccessible := 'False'; ExternalVisible := 'False'; ExternalWritable := 'False'} : Bool;
            xSpare_28 { ExternalAccessible := 'False'; ExternalVisible := 'False'; ExternalWritable := 'False'} : Bool;
            xSpare_29 { ExternalAccessible := 'False'; ExternalVisible := 'False'; ExternalWritable := 'False'} : Bool;
            xSpare_30 { ExternalAccessible := 'False'; ExternalVisible := 'False'; ExternalWritable := 'False'} : Bool;
            xSpare_31 { ExternalAccessible := 'False'; ExternalVisible := 'False'; ExternalWritable := 'False'} : Bool;
         END_STRUCT;
      END_STRUCT;
      tHMR { ExternalWritable := 'False'} : Struct   // HMI Read
         xSpare0 { ExternalWritable := 'False'} : Bool;   //
         xSpare1 { ExternalWritable := 'False'} : Bool;
         xSpare2 { ExternalWritable := 'False'} : Bool;
         xSpare3 { ExternalWritable := 'False'} : Bool;
         xSpare4 { ExternalWritable := 'False'} : Bool;
         xSpare5 { ExternalWritable := 'False'} : Bool;
         xSpare6 { ExternalWritable := 'False'} : Bool;
         xSpare7 { ExternalWritable := 'False'} : Bool;
         xSpare8 { ExternalWritable := 'False'} : Bool;
         xSpare9 { ExternalWritable := 'False'} : Bool;
         xSpare10 { ExternalWritable := 'False'} : Bool;
         xSpare11 { ExternalWritable := 'False'} : Bool;
         xSpare12 { ExternalWritable := 'False'} : Bool;
         xSpare13 { ExternalWritable := 'False'} : Bool;
         xSpare14 { ExternalWritable := 'False'} : Bool;   //
         xSpare15 { ExternalWritable := 'False'} : Bool;
         xSpare16 { ExternalWritable := 'False'} : Bool;
         xSpare17 { ExternalWritable := 'False'} : Bool;
         xSpare18 { ExternalWritable := 'False'} : Bool;
         xSpare19 { ExternalWritable := 'False'} : Bool;
         xSpare20 { ExternalWritable := 'False'} : Bool;
         xSpare21 { ExternalWritable := 'False'} : Bool;
         xSpare22 { ExternalWritable := 'False'} : Bool;
         xSpare23 { ExternalWritable := 'False'} : Bool;
         xSpare24 { ExternalWritable := 'False'} : Bool;
         xSpare25 { ExternalWritable := 'False'} : Bool;
         xSpare26 { ExternalWritable := 'False'} : Bool;
         xSpare27 { ExternalWritable := 'False'} : Bool;
         xSpare28 { ExternalWritable := 'False'} : Bool;
         xSpare29 { ExternalWritable := 'False'} : Bool;
         xSpare30 { ExternalWritable := 'False'} : Bool;
         xSpare31 { ExternalWritable := 'False'} : Bool;
         xSpare { ExternalWritable := 'False'} : Array[0..15] of Bool;
         iSpare0 { ExternalWritable := 'False'} : Int;
         iSpare1 { ExternalWritable := 'False'} : Int;
         iSpare2 { ExternalWritable := 'False'} : Int;
         iSpare3 { ExternalWritable := 'False'} : Int;
         iSpare4 { ExternalWritable := 'False'} : Int;
         iSpare5 { ExternalWritable := 'False'} : Int;
         iSpare6 { ExternalWritable := 'False'} : Int;
         iSpare7 { ExternalWritable := 'False'} : Int;
         iSpare8 { ExternalWritable := 'False'} : Int;
         iSpare9 { ExternalWritable := 'False'} : Int;
         iSpare10 { ExternalWritable := 'False'} : Int;
         iSpare11 { ExternalWritable := 'False'} : Int;
         iSpare12 { ExternalWritable := 'False'} : Int;
         iSpare13 { ExternalWritable := 'False'} : Int;
         iSpare14 { ExternalWritable := 'False'} : Int;
         iSpare15 { ExternalWritable := 'False'} : Int;
         iSpare16 { ExternalWritable := 'False'} : Int;
         dDistanceSnaproll_cmm { ExternalWritable := 'False'} : DInt;   // Distance from snaproll [mm/100] {mm/100|mm|x|x|M}
         dCameraStatus { ExternalWritable := 'False'} : DInt;   // Camera status (1=Disabled, 3=Enabled, 7=Anomaly) {x|x|x|x|O}
         dSpare2 { ExternalWritable := 'False'} : DInt;   // Distance from center line [mm/100] {mm/100|mm|X|X|O}
         dCurrentGrossWidth_cmm { ExternalWritable := 'False'} : DInt;   // Gross width [mm/100] {mm/100|mm|X|X|O}
         dCurrentNetWidth_cmm { ExternalWritable := 'False'} : DInt;   // Net width [mm/100] {mm/100|mm|X|X|O}
         dCurrentGrossWander_cmm { ExternalWritable := 'False'} : DInt;   // Gross wander [mm/100] {mm/100|mm|X|X|O}
         dCurrentNetWander_cmm { ExternalWritable := 'False'} : DInt;   // Net wander [mm/100] {mm/100|mm|X|X|O}
         dSpare7 { ExternalWritable := 'False'} : DInt;
         dSpare8 { ExternalWritable := 'False'} : DInt;
         dSpare9 { ExternalWritable := 'False'} : DInt;
         dSpare10 { ExternalWritable := 'False'} : DInt;
         dSpare11 { ExternalWritable := 'False'} : DInt;
         dSpare12 { ExternalWritable := 'False'} : DInt;
         dSpare13 { ExternalWritable := 'False'} : DInt;
         dSpare14 { ExternalWritable := 'False'} : DInt;
         dSpare15 { ExternalWritable := 'False'} : DInt;
         rSpare0 { ExternalWritable := 'False'} : Real;
         rSpare1 { ExternalWritable := 'False'} : Real;
         rSpare2 { ExternalWritable := 'False'} : Real;
         rSpare3 { ExternalWritable := 'False'} : Real;
         rSpare4 { ExternalWritable := 'False'} : Real;
         rSpare5 { ExternalWritable := 'False'} : Real;
         rSpare6 { ExternalWritable := 'False'} : Real;
         rSpare7 { ExternalWritable := 'False'} : Real;
         rSpare8 { ExternalWritable := 'False'} : Real;
         tManCmd { ExternalWritable := 'False'} : Struct
            xSpare1 { ExternalWritable := 'False'} : Bool;   //
            xSpare2 { ExternalWritable := 'False'} : Bool;
            xSpare3 { ExternalWritable := 'False'} : Bool;
            xSpare4 { ExternalWritable := 'False'} : Bool;
            xSpare5 { ExternalWritable := 'False'} : Bool;
            xSpare6 { ExternalWritable := 'False'} : Bool;
            xSpare7 { ExternalWritable := 'False'} : Bool;
            xSpare8 { ExternalWritable := 'False'} : Bool;
            xSpare9 { ExternalWritable := 'False'} : Bool;
            xSpare10 { ExternalWritable := 'False'} : Bool;
            xSpare11 { ExternalWritable := 'False'} : Bool;
            xSpare12 { ExternalWritable := 'False'} : Bool;
            xSpare13 { ExternalWritable := 'False'} : Bool;
            xSpare14 { ExternalWritable := 'False'} : Bool;
            xSpare15 { ExternalWritable := 'False'} : Bool;
            xSpare { ExternalWritable := 'False'} : Array[0..15] of Bool;
         END_STRUCT;
      END_STRUCT;
      tHMW : Struct   // HMI Write
         xSpare0 { ExternalWritable := 'False'} : Bool;
         xSpare1 : Bool;
         xSpare2 : Bool;
         xSpare3 : Bool;
         xSpare4 : Bool;
         xSpare5 : Bool;
         xSpare6 : Bool;
         xSpare7 : Bool;
         xSpare8 : Bool;
         xSpare9 : Bool;
         xSpare10 : Bool;
         xSpare11 : Bool;
         xSpare12 : Bool;
         xSpare13 : Bool;
         xSpare14 : Bool;   //
         xUpdateDistanceSnaproll : Bool;   // Update distance from snaproll {x|x|x|x|M}
         xSpare16 : Bool;   //
         xSpare17 : Bool;   //
         xSpare18 : Bool;
         xSpare19 : Bool;
         xSpare20 : Bool;
         xSpare21 : Bool;
         xSpare22 : Bool;
         xSpare23 : Bool;
         xSpare24 : Bool;
         xSpare25 : Bool;
         xSpare26 : Bool;
         xSpare27 : Bool;
         xSpare28 : Bool;
         xSpare29 : Bool;
         xSpare30 : Bool;
         xSpare31 : Bool;
         xSpare : Array[0..15] of Bool;
         iSpare0 : Int;
         iSpare1 : Int;
         iSpare2 : Int;
         iSpare3 : Int;
         iSpare4 : Int;
         iSpare5 : Int;
         iSpare6 : Int;
         iSpare7 : Int;
         iSpare8 : Int;
         iSpare9 : Int;
         iSpare10 : Int;
         iSpare11 : Int;
         iSpare12 : Int;
         iSpare13 : Int;
         iSpare14 : Int;
         iSpare15 : Int;
         iSpare16 : Int;
         dDistanceSnaproll_cmm : DInt;   // Distance from snaproll [mm/100] {mm/100|mm|1|70000|M}
         dSpare1 : DInt;
         dSpare2 : DInt;
         dSpare3 : DInt;
         dSpare4 : DInt;
         dSpare5 : DInt;
         dSpare6 : DInt;
         dSpare7 : DInt;
         dSpare8 : DInt;
         dSpare9 : DInt;
         dSpare10 : DInt;
         dSpare11 : DInt;
         dSpare12 : DInt;
         dSpare13 : DInt;
         dSpare14 : DInt;
         dSpare15 : DInt;
         dSpare16 : DInt;
         rSpare0 : Real;
         rSpare1 : Real;
         rSpare2 : Real;
         rSpare3 : Real;
         rSpare4 : Real;
         rSpare5 : Real;
         rSpare6 : Real;
         rSpare7 : Real;
         rSpare8 : Real;
         tManCmd : Struct
            xFanCommand : Bool;   // Fan command {x|x|x|x|O}
            xSpare1 : Bool;   //
            xSpare2 : Bool;
            xSpare3 : Bool;
            xSpare4 : Bool;
            xSpare5 : Bool;
            xSpare6 : Bool;
            xSpare7 : Bool;
            xSpare8 : Bool;
            xSpare9 : Bool;
            xSpare10 : Bool;
            xSpare11 : Bool;
            xSpare12 : Bool;
            xSpare13 : Bool;
            xSpare14 : Bool;
            xSpare15 : Bool;
            xSpare16 : Bool;
            xSpare17 : Bool;
            xSpare18 : Bool;
            xSpare19 : Bool;
            xSpare20 : Bool;
            xSpare21 : Bool;
            xSpare22 : Bool;
            xSpare23 : Bool;
            xSpare24 : Bool;
            xSpare25 : Bool;
            xSpare26 : Bool;
            xSpare27 : Bool;
            xSpare28 : Bool;
            xSpare29 : Bool;
            xSpare30 : Bool;
            xSpare31 : Bool;
         END_STRUCT;
      END_STRUCT;
   END_STRUCT;


BEGIN
   tHMR.dCameraStatus := 0;
   tHMW.tManCmd.xSpare1 := false;

END_DATA_BLOCK

DATA_BLOCK "DB_MAN_INSP_HMI"
{ DB_Accessible_From_OPC_UA := 'FALSE' ;
 DB_Accessible_From_Webserver := 'FALSE' ;
 S7_Optimized_Access := 'FALSE' }
VERSION : 0.1
NON_RETAIN
   STRUCT
      tALM { ExternalWritable := 'False'} : Struct   // HMI Alarms
         tE { ExternalWritable := 'False'} : Struct   // Stopping faults
            xSpare_0 { ExternalWritable := 'False'} : Bool;
            xSpare_1 { ExternalWritable := 'False'} : Bool;
            xSpare_2 { ExternalWritable := 'False'} : Bool;
            xSpare_3 { ExternalWritable := 'False'} : Bool;
            xSpare_4 { ExternalWritable := 'False'} : Bool;
            xSpare_5 { ExternalWritable := 'False'} : Bool;
            xSpare_6 { ExternalWritable := 'False'} : Bool;
            xSpare_7 { ExternalWritable := 'False'} : Bool;
            xSpare_8 { ExternalWritable := 'False'} : Bool;
            xSpare_9 { ExternalWritable := 'False'} : Bool;
            xSpare_10 { ExternalWritable := 'False'} : Bool;
            xSpare_11 { ExternalWritable := 'False'} : Bool;
            xSpare_12 { ExternalWritable := 'False'} : Bool;
            xSpare_13 { ExternalWritable := 'False'} : Bool;
            xSpare_14 { ExternalWritable := 'False'} : Bool;
            xSpare_15 { ExternalWritable := 'False'} : Bool;
            xSpare_16 { ExternalWritable := 'False'} : Bool;
            xSpare_17 { ExternalWritable := 'False'} : Bool;
            xSpare_18 { ExternalWritable := 'False'} : Bool;
            xSpare_19 { ExternalWritable := 'False'} : Bool;
            xSpare_20 { ExternalWritable := 'False'} : Bool;
            xSpare_21 { ExternalWritable := 'False'} : Bool;
            xSpare_22 { ExternalWritable := 'False'} : Bool;
            xSpare_23 { ExternalWritable := 'False'} : Bool;
            xSpare_24 { ExternalWritable := 'False'} : Bool;
            xSpare_25 { ExternalWritable := 'False'} : Bool;
            xSpare_26 { ExternalWritable := 'False'} : Bool;
            xSpare_27 { ExternalWritable := 'False'} : Bool;
            xSpare_28 { ExternalWritable := 'False'} : Bool;
            xSpare_29 { ExternalWritable := 'False'} : Bool;
            xSpare_30 { ExternalWritable := 'False'} : Bool;
            xSpare_31 { ExternalWritable := 'False'} : Bool;
         END_STRUCT;
         tS { ExternalWritable := 'False'} : Struct   // Stopping faults machine
            xPowerSupplyControl { ExternalWritable := 'False'} : Bool;   // NU.1A222/1L+.Power supply control {X|X|X|X|O}
            xSpare_1 { ExternalAccessible := 'False'; ExternalVisible := 'False'; ExternalWritable := 'False'} : Bool;
            xSpare_2 { ExternalAccessible := 'False'; ExternalVisible := 'False'; ExternalWritable := 'False'} : Bool;
            xSpare_3 { ExternalAccessible := 'False'; ExternalVisible := 'False'; ExternalWritable := 'False'} : Bool;
            xSpare_4 { ExternalAccessible := 'False'; ExternalVisible := 'False'; ExternalWritable := 'False'} : Bool;
            xSpare_5 { ExternalAccessible := 'False'; ExternalVisible := 'False'; ExternalWritable := 'False'} : Bool;
            xSpare_6 { ExternalAccessible := 'False'; ExternalVisible := 'False'; ExternalWritable := 'False'} : Bool;
            xSpare_7 { ExternalAccessible := 'False'; ExternalVisible := 'False'; ExternalWritable := 'False'} : Bool;
            xSpare_8 { ExternalAccessible := 'False'; ExternalVisible := 'False'; ExternalWritable := 'False'} : Bool;
            xSpare_9 { ExternalAccessible := 'False'; ExternalVisible := 'False'; ExternalWritable := 'False'} : Bool;
            xSpare_10 { ExternalAccessible := 'False'; ExternalVisible := 'False'; ExternalWritable := 'False'} : Bool;
            xSpare_11 { ExternalAccessible := 'False'; ExternalVisible := 'False'; ExternalWritable := 'False'} : Bool;
            xSpare_12 { ExternalAccessible := 'False'; ExternalVisible := 'False'; ExternalWritable := 'False'} : Bool;
            xSpare_13 { ExternalAccessible := 'False'; ExternalVisible := 'False'; ExternalWritable := 'False'} : Bool;
            xSpare_14 { ExternalAccessible := 'False'; ExternalVisible := 'False'; ExternalWritable := 'False'} : Bool;
            xSpare_15 { ExternalAccessible := 'False'; ExternalVisible := 'False'; ExternalWritable := 'False'} : Bool;
            xSpare_16 { ExternalAccessible := 'False'; ExternalVisible := 'False'; ExternalWritable := 'False'} : Bool;
            xSpare_17 { ExternalAccessible := 'False'; ExternalVisible := 'False'; ExternalWritable := 'False'} : Bool;
            xSpare_18 { ExternalAccessible := 'False'; ExternalVisible := 'False'; ExternalWritable := 'False'} : Bool;
            xSpare_19 { ExternalAccessible := 'False'; ExternalVisible := 'False'; ExternalWritable := 'False'} : Bool;
            xSpare_20 { ExternalAccessible := 'False'; ExternalVisible := 'False'; ExternalWritable := 'False'} : Bool;
            xSpare_21 { ExternalAccessible := 'False'; ExternalVisible := 'False'; ExternalWritable := 'False'} : Bool;
            xSpare_22 { ExternalAccessible := 'False'; ExternalVisible := 'False'; ExternalWritable := 'False'} : Bool;
            xSpare_23 { ExternalAccessible := 'False'; ExternalVisible := 'False'; ExternalWritable := 'False'} : Bool;
            xSpare_24 { ExternalAccessible := 'False'; ExternalVisible := 'False'; ExternalWritable := 'False'} : Bool;
            xSpare_25 { ExternalAccessible := 'False'; ExternalVisible := 'False'; ExternalWritable := 'False'} : Bool;
            xSpare_26 { ExternalAccessible := 'False'; ExternalVisible := 'False'; ExternalWritable := 'False'} : Bool;
            xSpare_27 { ExternalAccessible := 'False'; ExternalVisible := 'False'; ExternalWritable := 'False'} : Bool;
            xSpare_28 { ExternalAccessible := 'False'; ExternalVisible := 'False'; ExternalWritable := 'False'} : Bool;
            xSpare_29 { ExternalAccessible := 'False'; ExternalVisible := 'False'; ExternalWritable := 'False'} : Bool;
            xSpare_30 { ExternalAccessible := 'False'; ExternalVisible := 'False'; ExternalWritable := 'False'} : Bool;
            xSpare_31 { ExternalAccessible := 'False'; ExternalVisible := 'False'; ExternalWritable := 'False'} : Bool;
         END_STRUCT;
         tF { ExternalAccessible := 'False'; ExternalVisible := 'False'; ExternalWritable := 'False'} : Struct   // Faults
            xSpare_0 { ExternalAccessible := 'False'; ExternalVisible := 'False'; ExternalWritable := 'False'} : Bool;
            xSpare_1 { ExternalAccessible := 'False'; ExternalVisible := 'False'; ExternalWritable := 'False'} : Bool;
            xSpare_2 { ExternalAccessible := 'False'; ExternalVisible := 'False'; ExternalWritable := 'False'} : Bool;
            xSpare_3 { ExternalAccessible := 'False'; ExternalVisible := 'False'; ExternalWritable := 'False'} : Bool;
            xSpare_4 { ExternalAccessible := 'False'; ExternalVisible := 'False'; ExternalWritable := 'False'} : Bool;
            xSpare_5 { ExternalAccessible := 'False'; ExternalVisible := 'False'; ExternalWritable := 'False'} : Bool;
            xSpare_6 { ExternalAccessible := 'False'; ExternalVisible := 'False'; ExternalWritable := 'False'} : Bool;
            xSpare_7 { ExternalAccessible := 'False'; ExternalVisible := 'False'; ExternalWritable := 'False'} : Bool;
            xSpare_8 { ExternalAccessible := 'False'; ExternalVisible := 'False'; ExternalWritable := 'False'} : Bool;
            xSpare_9 { ExternalAccessible := 'False'; ExternalVisible := 'False'; ExternalWritable := 'False'} : Bool;
            xSpare_10 { ExternalAccessible := 'False'; ExternalVisible := 'False'; ExternalWritable := 'False'} : Bool;
            xSpare_11 { ExternalAccessible := 'False'; ExternalVisible := 'False'; ExternalWritable := 'False'} : Bool;
            xSpare_12 { ExternalAccessible := 'False'; ExternalVisible := 'False'; ExternalWritable := 'False'} : Bool;
            xSpare_13 { ExternalAccessible := 'False'; ExternalVisible := 'False'; ExternalWritable := 'False'} : Bool;
            xSpare_14 { ExternalAccessible := 'False'; ExternalVisible := 'False'; ExternalWritable := 'False'} : Bool;
            xSpare_15 { ExternalAccessible := 'False'; ExternalVisible := 'False'; ExternalWritable := 'False'} : Bool;
            xSpare_16 { ExternalAccessible := 'False'; ExternalVisible := 'False'; ExternalWritable := 'False'} : Bool;
            xSpare_17 { ExternalAccessible := 'False'; ExternalVisible := 'False'; ExternalWritable := 'False'} : Bool;
            xSpare_18 { ExternalAccessible := 'False'; ExternalVisible := 'False'; ExternalWritable := 'False'} : Bool;
            xSpare_19 { ExternalAccessible := 'False'; ExternalVisible := 'False'; ExternalWritable := 'False'} : Bool;
            xSpare_20 { ExternalAccessible := 'False'; ExternalVisible := 'False'; ExternalWritable := 'False'} : Bool;
            xSpare_21 { ExternalAccessible := 'False'; ExternalVisible := 'False'; ExternalWritable := 'False'} : Bool;
            xSpare_22 { ExternalAccessible := 'False'; ExternalVisible := 'False'; ExternalWritable := 'False'} : Bool;
            xSpare_23 { ExternalAccessible := 'False'; ExternalVisible := 'False'; ExternalWritable := 'False'} : Bool;
            xSpare_24 { ExternalAccessible := 'False'; ExternalVisible := 'False'; ExternalWritable := 'False'} : Bool;
            xSpare_25 { ExternalAccessible := 'False'; ExternalVisible := 'False'; ExternalWritable := 'False'} : Bool;
            xSpare_26 { ExternalAccessible := 'False'; ExternalVisible := 'False'; ExternalWritable := 'False'} : Bool;
            xSpare_27 { ExternalAccessible := 'False'; ExternalVisible := 'False'; ExternalWritable := 'False'} : Bool;
            xSpare_28 { ExternalAccessible := 'False'; ExternalVisible := 'False'; ExternalWritable := 'False'} : Bool;
            xSpare_29 { ExternalAccessible := 'False'; ExternalVisible := 'False'; ExternalWritable := 'False'} : Bool;
            xSpare_30 { ExternalAccessible := 'False'; ExternalVisible := 'False'; ExternalWritable := 'False'} : Bool;
            xSpare_31 { ExternalAccessible := 'False'; ExternalVisible := 'False'; ExternalWritable := 'False'} : Bool;
         END_STRUCT;
         tW { ExternalAccessible := 'False'; ExternalVisible := 'False'; ExternalWritable := 'False'} : Struct   // Warnings
            xSpare_0 { ExternalAccessible := 'False'; ExternalVisible := 'False'; ExternalWritable := 'False'} : Bool;
            xSpare_1 { ExternalAccessible := 'False'; ExternalVisible := 'False'; ExternalWritable := 'False'} : Bool;
            xSpare_2 { ExternalAccessible := 'False'; ExternalVisible := 'False'; ExternalWritable := 'False'} : Bool;
            xSpare_3 { ExternalAccessible := 'False'; ExternalVisible := 'False'; ExternalWritable := 'False'} : Bool;
            xSpare_4 { ExternalAccessible := 'False'; ExternalVisible := 'False'; ExternalWritable := 'False'} : Bool;
            xSpare_5 { ExternalAccessible := 'False'; ExternalVisible := 'False'; ExternalWritable := 'False'} : Bool;
            xSpare_6 { ExternalAccessible := 'False'; ExternalVisible := 'False'; ExternalWritable := 'False'} : Bool;
            xSpare_7 { ExternalAccessible := 'False'; ExternalVisible := 'False'; ExternalWritable := 'False'} : Bool;
            xSpare_8 { ExternalAccessible := 'False'; ExternalVisible := 'False'; ExternalWritable := 'False'} : Bool;
            xSpare_9 { ExternalAccessible := 'False'; ExternalVisible := 'False'; ExternalWritable := 'False'} : Bool;
            xSpare_10 { ExternalAccessible := 'False'; ExternalVisible := 'False'; ExternalWritable := 'False'} : Bool;
            xSpare_11 { ExternalAccessible := 'False'; ExternalVisible := 'False'; ExternalWritable := 'False'} : Bool;
            xSpare_12 { ExternalAccessible := 'False'; ExternalVisible := 'False'; ExternalWritable := 'False'} : Bool;
            xSpare_13 { ExternalAccessible := 'False'; ExternalVisible := 'False'; ExternalWritable := 'False'} : Bool;
            xSpare_14 { ExternalAccessible := 'False'; ExternalVisible := 'False'; ExternalWritable := 'False'} : Bool;
            xSpare_15 { ExternalAccessible := 'False'; ExternalVisible := 'False'; ExternalWritable := 'False'} : Bool;
            xSpare_16 { ExternalAccessible := 'False'; ExternalVisible := 'False'; ExternalWritable := 'False'} : Bool;
            xSpare_17 { ExternalAccessible := 'False'; ExternalVisible := 'False'; ExternalWritable := 'False'} : Bool;
            xSpare_18 { ExternalAccessible := 'False'; ExternalVisible := 'False'; ExternalWritable := 'False'} : Bool;
            xSpare_19 { ExternalAccessible := 'False'; ExternalVisible := 'False'; ExternalWritable := 'False'} : Bool;
            xSpare_20 { ExternalAccessible := 'False'; ExternalVisible := 'False'; ExternalWritable := 'False'} : Bool;
            xSpare_21 { ExternalAccessible := 'False'; ExternalVisible := 'False'; ExternalWritable := 'False'} : Bool;
            xSpare_22 { ExternalAccessible := 'False'; ExternalVisible := 'False'; ExternalWritable := 'False'} : Bool;
            xSpare_23 { ExternalAccessible := 'False'; ExternalVisible := 'False'; ExternalWritable := 'False'} : Bool;
            xSpare_24 { ExternalAccessible := 'False'; ExternalVisible := 'False'; ExternalWritable := 'False'} : Bool;
            xSpare_25 { ExternalAccessible := 'False'; ExternalVisible := 'False'; ExternalWritable := 'False'} : Bool;
            xSpare_26 { ExternalAccessible := 'False'; ExternalVisible := 'False'; ExternalWritable := 'False'} : Bool;
            xSpare_27 { ExternalAccessible := 'False'; ExternalVisible := 'False'; ExternalWritable := 'False'} : Bool;
            xSpare_28 { ExternalAccessible := 'False'; ExternalVisible := 'False'; ExternalWritable := 'False'} : Bool;
            xSpare_29 { ExternalAccessible := 'False'; ExternalVisible := 'False'; ExternalWritable := 'False'} : Bool;
            xSpare_30 { ExternalAccessible := 'False'; ExternalVisible := 'False'; ExternalWritable := 'False'} : Bool;
            xSpare_31 { ExternalAccessible := 'False'; ExternalVisible := 'False'; ExternalWritable := 'False'} : Bool;
         END_STRUCT;
      END_STRUCT;
      tHMR { ExternalWritable := 'False'} : Struct   // HMI Read
         xSpare0 { ExternalWritable := 'False'} : Bool;
         xSpare1 { ExternalWritable := 'False'} : Bool;
         xSpare2 { ExternalWritable := 'False'} : Bool;
         xSpare3 { ExternalWritable := 'False'} : Bool;
         xSpare4 { ExternalWritable := 'False'} : Bool;
         xSpare5 { ExternalWritable := 'False'} : Bool;
         xSpare6 { ExternalWritable := 'False'} : Bool;
         xSpare7 { ExternalWritable := 'False'} : Bool;
         xSpare8 { ExternalWritable := 'False'} : Bool;
         xSpare9 { ExternalWritable := 'False'} : Bool;
         xSpare10 { ExternalWritable := 'False'} : Bool;
         xSpare11 { ExternalWritable := 'False'} : Bool;
         xSpare12 { ExternalWritable := 'False'} : Bool;
         xSpare13 { ExternalWritable := 'False'} : Bool;
         xManualCommandEnabled { ExternalWritable := 'False'} : Bool;   // Manual Command enabled {x|x|x|x|O}
         xSpare15 { ExternalWritable := 'False'} : Bool;
         xSpare16 { ExternalWritable := 'False'} : Bool;
         xSpare17 { ExternalWritable := 'False'} : Bool;
         xSpare18 { ExternalWritable := 'False'} : Bool;
         xSpare19 { ExternalWritable := 'False'} : Bool;
         xSpare20 { ExternalWritable := 'False'} : Bool;
         xSpare21 { ExternalWritable := 'False'} : Bool;
         xSpare22 { ExternalWritable := 'False'} : Bool;
         xSpare23 { ExternalWritable := 'False'} : Bool;
         xSpare24 { ExternalWritable := 'False'} : Bool;
         xSpare25 { ExternalWritable := 'False'} : Bool;
         xSpare26 { ExternalWritable := 'False'} : Bool;
         xSpare27 { ExternalWritable := 'False'} : Bool;
         xSpare28 { ExternalWritable := 'False'} : Bool;
         xSpare29 { ExternalWritable := 'False'} : Bool;
         xSpare30 { ExternalWritable := 'False'} : Bool;
         xSpare31 { ExternalWritable := 'False'} : Bool;
         xSpare { ExternalWritable := 'False'} : Array[0..15] of Bool;
         iSpare0 { ExternalWritable := 'False'} : Int;
         iSpare1 { ExternalWritable := 'False'} : Int;
         iSpare2 { ExternalWritable := 'False'} : Int;
         iSpare3 { ExternalWritable := 'False'} : Int;
         iSpare4 { ExternalWritable := 'False'} : Int;
         iSpare5 { ExternalWritable := 'False'} : Int;
         iSpare6 { ExternalWritable := 'False'} : Int;
         iSpare7 { ExternalWritable := 'False'} : Int;
         iSpare8 { ExternalWritable := 'False'} : Int;
         iSpare9 { ExternalWritable := 'False'} : Int;
         iSpare10 { ExternalWritable := 'False'} : Int;
         iSpare11 { ExternalWritable := 'False'} : Int;
         iSpare12 { ExternalWritable := 'False'} : Int;
         iSpare13 { ExternalWritable := 'False'} : Int;
         iSpare14 { ExternalWritable := 'False'} : Int;
         iSpare15 { ExternalWritable := 'False'} : Int;
         iSpare16 { ExternalWritable := 'False'} : Int;
         dDistanceSnaproll_cmm { ExternalWritable := 'False'} : DInt;   // Distance from snaproll [mm/100] {mm/100|mm|x|x|M}
         dSpare1 { ExternalWritable := 'False'} : DInt;
         dSpare2 { ExternalWritable := 'False'} : DInt;
         dSpare3 { ExternalWritable := 'False'} : DInt;
         dSpare4 { ExternalWritable := 'False'} : DInt;
         dSpare5 { ExternalWritable := 'False'} : DInt;
         dSpare6 { ExternalWritable := 'False'} : DInt;
         dSpare7 { ExternalWritable := 'False'} : DInt;
         dSpare8 { ExternalWritable := 'False'} : DInt;
         dSpare9 { ExternalWritable := 'False'} : DInt;
         dSpare10 { ExternalWritable := 'False'} : DInt;
         dSpare11 { ExternalWritable := 'False'} : DInt;
         dSpare12 { ExternalWritable := 'False'} : DInt;
         dSpare13 { ExternalWritable := 'False'} : DInt;
         dSpare14 { ExternalWritable := 'False'} : DInt;
         dSpare15 { ExternalWritable := 'False'} : DInt;
         rSpare0 { ExternalWritable := 'False'} : Real;
         rSpare1 { ExternalWritable := 'False'} : Real;
         rSpare2 { ExternalWritable := 'False'} : Real;
         rSpare3 { ExternalWritable := 'False'} : Real;
         rSpare4 { ExternalWritable := 'False'} : Real;
         rSpare5 { ExternalWritable := 'False'} : Real;
         rSpare6 { ExternalWritable := 'False'} : Real;
         rSpare7 { ExternalWritable := 'False'} : Real;
         rSpare8 { ExternalWritable := 'False'} : Real;
         tManCmd { ExternalWritable := 'False'} : Struct
            xSpare0 { ExternalWritable := 'False'} : Bool;
            xSpare1 { ExternalWritable := 'False'} : Bool;   //
            xSpare2 { ExternalWritable := 'False'} : Bool;
            xSpare3 { ExternalWritable := 'False'} : Bool;
            xSpare4 { ExternalWritable := 'False'} : Bool;
            xSpare5 { ExternalWritable := 'False'} : Bool;
            xSpare6 { ExternalWritable := 'False'} : Bool;
            xSpare7 { ExternalWritable := 'False'} : Bool;
            xSpare8 { ExternalWritable := 'False'} : Bool;
            xSpare9 { ExternalWritable := 'False'} : Bool;
            xSpare10 { ExternalWritable := 'False'} : Bool;
            xSpare11 { ExternalWritable := 'False'} : Bool;
            xSpare12 { ExternalWritable := 'False'} : Bool;
            xSpare13 { ExternalWritable := 'False'} : Bool;
            xSpare14 { ExternalWritable := 'False'} : Bool;
            xSpare15 { ExternalWritable := 'False'} : Bool;
            xSpare { ExternalWritable := 'False'} : Array[0..15] of Bool;
         END_STRUCT;
      END_STRUCT;
      tHMW : Struct   // HMI Write
         xSpare0 : Bool;   //
         xSpare1 : Bool;
         xSpare2 : Bool;
         xSpare3 : Bool;
         xSpare4 : Bool;
         xSpare5 : Bool;
         xSpare6 : Bool;
         xSpare7 : Bool;
         "xEnabledContinuosDef[0]" : Bool;   // Enable continuos defect {x|x|x|x|O}
         "xEnabledContinuosDef[1]" : Bool;   // Enable continuos defect {x|x|x|x|O}
         "xEnabledContinuosDef[2]" : Bool;   // Enable continuos defect {x|x|x|x|O}
         "xEnabledContinuosDef[3]" : Bool;   // Enable continuos defect {x|x|x|x|O}
         xSpare12 : Bool;
         xSpare13 : Bool;
         xEnableManualCommand : Bool;   // Enable Disable Manual command {x|x|x|x|O}
         xUpdateDistanceSnaproll : Bool;   // Update distance from snaproll {x|x|x|x|M}
         xDefectCalibration : Bool;   // Calibration.Calibrate defect {x|x|x|x|M}
         xSpare17 : Bool;
         xSpare18 : Bool;
         xSpare19 : Bool;
         xSpare20 : Bool;
         xSpare21 : Bool;
         xSpare22 : Bool;
         xSpare23 : Bool;
         xSpare24 : Bool;
         xSpare25 : Bool;
         xSpare26 : Bool;
         xSpare27 : Bool;
         xSpare28 : Bool;
         xSpare29 : Bool;
         xSpare30 : Bool;
         xSpare31 : Bool;
         xSpare : Array[0..15] of Bool;
         iSpare0 : Int;
         iSpare1 : Int;
         iSpare2 : Int;
         iSpare3 : Int;
         iSpare4 : Int;
         iSpare5 : Int;
         iSpare6 : Int;
         iSpare7 : Int;
         iSpare8 : Int;
         iSpare9 : Int;
         iSpare10 : Int;
         iSpare11 : Int;
         iSpare12 : Int;
         iSpare13 : Int;
         iSpare14 : Int;
         iSpare15 : Int;
         iSpare16 : Int;
         dDistanceSnaproll_cmm : DInt;   // Distance from snaproll [mm/100] {mm/100|mm|1|70000|M}
         dDefectLength_cmm : DInt;   // Defect length [mm/100] {mm/100|mm|1|1000|O}
         dDefectWidth_cmm : DInt;   // Defect width [mm/100] {mm/100|mm|1|1000|O}
         dCalibDefectTheoPosX_cmm : DInt;   // Calibration. Theorical defect position X [mm/100] {mm/100|mm|1|7000|O}
         dCalibDefectRealPosX_cmm : DInt;   // Calibration. Real defect position X  [mm/100] {mm/100|mm|1|7000|O}
         "dButtonClass[0]" : DInt;   // Buttons defect class {x|x|1|20|O}
         "dButtonClass[1]" : DInt;   // Buttons defect class {x|x|1|20|O}
         "dButtonClass[2]" : DInt;   // Buttons defect class {x|x|1|20|O}
         "dButtonClass[3]" : DInt;   // Buttons defect class {x|x|1|20|O}
         "dButtonPosition_cmm[0]" : DInt;   // Buttons defect position {mm/100|mm|-3000|3000|O}
         "dButtonPosition_cmm[1]" : DInt;   // Buttons defect position {mm/100|mm|-3000|3000|O}
         "dButtonPosition_cmm[2]" : DInt;   // Buttons defect position {mm/100|mm|-3000|3000|O}
         "dButtonPosition_cmm[3]" : DInt;   // Buttons defect position {mm/100|mm|-3000|3000|O}
         dSpare13 : DInt;
         dSpare14 : DInt;
         dSpare15 : DInt;
         dSpare16 : DInt;
         rSpare0 : Real;
         rSpare1 : Real;
         rSpare2 : Real;
         rSpare3 : Real;
         rSpare4 : Real;
         rSpare5 : Real;
         rSpare6 : Real;
         rSpare7 : Real;
         rSpare8 : Real;
         tManCmd : Struct
            xSpare0 : Bool;   //
            xSpare1 : Bool;   //
            xSpare2 { ExternalWritable := 'False'} : Bool;
            xSpare3 { ExternalWritable := 'False'} : Bool;
            xSpare4 { ExternalWritable := 'False'} : Bool;
            xSpare5 { ExternalWritable := 'False'} : Bool;
            xSpare6 { ExternalWritable := 'False'} : Bool;
            xSpare7 { ExternalWritable := 'False'} : Bool;
            xSpare8 { ExternalWritable := 'False'} : Bool;
            xSpare9 { ExternalWritable := 'False'} : Bool;
            xSpare10 { ExternalWritable := 'False'} : Bool;
            xSpare11 { ExternalWritable := 'False'} : Bool;
            xSpare12 { ExternalWritable := 'False'} : Bool;
            xSpare13 { ExternalWritable := 'False'} : Bool;
            xSpare14 { ExternalWritable := 'False'} : Bool;
            xSpare15 { ExternalWritable := 'False'} : Bool;
            xSpare16 : Bool;
            xSpare17 : Bool;
            xSpare18 : Bool;
            xSpare19 : Bool;
            xSpare20 : Bool;
            xSpare21 : Bool;
            xSpare22 : Bool;
            xSpare23 : Bool;
            xSpare24 : Bool;
            xSpare25 : Bool;
            xSpare26 : Bool;
            xSpare27 : Bool;
            xSpare28 : Bool;
            xSpare29 : Bool;
            xSpare30 : Bool;
            xSpare31 : Bool;
         END_STRUCT;
      END_STRUCT;
   END_STRUCT;


BEGIN
   tHMW.tManCmd.xSpare1 := false;

END_DATA_BLOCK

